  MoveL 4549 to (447.41, 537.05, 80) mm, rotated rx -180 ry 0 rz 160 deg; joints [12.233, 59.659, 9.495, -145.993, 72.482, 168.52]
  Set speed (17.8 mm/s)
  Call Extruder(266.02941)
  MoveL 4550 to (446.66, 535.95, 80) mm, rotated rx -180 ry 0 rz 160 deg; joints [12.104, 59.545, 9.763, -146.152, 72.584, 168.65]
  Call Extruder(270.12831)
  MoveL 4551 to (445.95, 534.87, 80) mm, rotated rx 180 ry 0 rz 160 deg; joints [11.975, 59.436, 10.019, -146.31, 72.681, 168.775]
  Set speed (17.8 mm/s)
  Call Extruder(274.24674)
  MoveL 4552 to (445.25, 533.77, 80) mm, rotated rx 180 ry 0 rz 160 deg; joints [11.843, 59.33, 10.27, -146.471, 72.776, 168.899]
  Call Extruder(278.37060)
  MoveL 4553 to (444.58, 532.66, 80) mm, rotated rx -180 ry 0 rz 160 deg; joints [11.707, 59.226, 10.515, -146.634, 72.867, 169.022]
  Set speed (17.8 mm/s)
  Call Extruder(282.63092)
  MoveL 4554 to (443.91, 531.49, 80) mm, rotated rx 180 ry 0 rz 160 deg; joints [11.563, 59.122, 10.76, -146.806, 72.959, 169.146]
  Call Extruder(286.74153)
  MoveL 4555 to (443.28, 530.35, 80) mm, rotated rx -180 ry 0 rz 160 deg; joints [11.421, 59.025, 10.991, -146.974, 73.044, 169.265]
  Call Extruder(290.93893)
  MoveL 4556 to (442.67, 529.17, 80) mm, rotated rx 180 ry 0 rz 160 deg; joints [11.274, 58.929, 11.219, -147.147, 73.127, 169.384]
  Set speed (17.8 mm/s)
  Call Extruder(295.04718)
  MoveL 4557 to (442.09, 528.01, 80) mm, rotated rx 180 ry 0 rz 160 deg; joints [11.126, 58.838, 11.436, -147.32, 73.205, 169.499]
  Set speed (17.8 mm/s)
  Call Extruder(299.35678)
  MoveL 4558 to (441.52, 526.78, 80) mm, rotated rx 180 ry 0 rz 160 deg; joints [10.968, 58.746, 11.654, -147.503, 73.283, 169.617]
  Set speed (17.8 mm/s)
  Call Extruder(303.33927)
  MoveL 4559 to (441, 525.63, 80) mm, rotated rx 180 ry 0 rz 160 deg; joints [10.82, 58.663, 11.851, -147.673, 73.353, 169.725]
  Set speed (17.8 mm/s)
  Call Extruder(307.68159)
  MoveL 4560 to (440.47, 524.37, 80) mm, rotated rx 180 ry 0 rz 160 deg; joints [10.654, 58.577, 12.056, -147.862, 73.424, 169.839]
  Set speed (17.8 mm/s)
  Call Extruder(311.65960)
  MoveL 4561 to (440, 523.2, 80) mm, rotated rx 180 ry 0 rz 160 deg; joints [10.501, 58.5, 12.239, -148.036, 73.488, 169.943]
  Set speed (17.8 mm/s)
  Call Extruder(316.02784)
  MoveL 4562 to (439.53, 521.91, 80) mm, rotated rx 180 ry 0 rz 160 deg; joints [10.33, 58.421, 12.429, -148.229, 73.552, 170.054]
  Call Extruder(320.19544)
  MoveL 4563 to (439.08, 520.67, 80) mm, rotated rx -180 ry 0 rz 160 deg; joints [10.164, 58.347, 12.607, -148.415, 73.612, 170.159]
  Set speed (17.8 mm/s)
  Call Extruder(324.35507)
  MoveL 4564 to (438.68, 519.42, 80) mm, rotated rx 180 ry 0 rz 160 deg; joints [9.996, 58.278, 12.773, -148.603, 73.665, 170.26]
  Call Extruder(328.30973)
  MoveL 4565 to (438.31, 518.23, 80) mm, rotated rx -180 ry 0 rz 160 deg; joints [9.834, 58.213, 12.926, -148.782, 73.715, 170.355]
  Call Extruder(332.69708)
  MoveL 4566 to (437.94, 516.9, 80) mm, rotated rx 180 ry 0 rz 160 deg; joints [9.652, 58.147, 13.086, -148.984, 73.764, 170.458]
  Set speed (17.8 mm/s)
  Call Extruder(336.73190)
  MoveL 4567 to (437.61, 515.67, 80) mm, rotated rx 180 ry 0 rz 160 deg; joints [9.483, 58.088, 13.227, -149.17, 73.807, 170.55]
  Set speed (17.8 mm/s)
  Call Extruder(341.04868)
  MoveL 4568 to (437.3, 514.34, 80) mm, rotated rx -180 ry 0 rz 160 deg; joints [9.299, 58.03, 13.368, -149.371, 73.848, 170.647]
  Call Extruder(345.11422)
  MoveL 4569 to (437.02, 513.09, 80) mm, rotated rx -180 ry 0 rz 160 deg; joints [9.125, 57.977, 13.496, -149.561, 73.884, 170.736]
  Set speed (17.8 mm/s)
  Call Extruder(353.56410)
  MoveL 4570 to (436.53, 510.46, 80) mm, rotated rx 180 ry 0 rz 160 deg; joints [8.756, 57.878, 13.734, -149.96, 73.946, 170.914]
  Set speed (17.8 mm/s)
  Call Extruder(361.89397)
  MoveL 4571 to (436.15, 507.86, 80) mm, rotated rx 180 ry 0 rz 160 deg; joints [8.386, 57.794, 13.937, -150.358, 73.991, 171.081]
  Call Extruder(370.22374)
  MoveL 4572 to (435.89, 505.24, 80) mm, rotated rx -180 ry 0 rz 160 deg; joints [8.01, 57.724, 14.107, -150.758, 74.02, 171.238]
  Set speed (17.8 mm/s)
  Call Extruder(378.39440)
  MoveL 4573 to (435.73, 502.67, 80) mm, rotated rx -180 ry 0 rz 160 deg; joints [7.637, 57.668, 14.242, -151.153, 74.033, 171.384]
  Set speed (17.8 mm/s)
  Call Extruder(386.80288)
  MoveL 4574 to (435.67, 500.01, 80) mm, rotated rx 180 ry 0 rz 160 deg; joints [7.249, 57.624, 14.348, -151.56, 74.03, 171.524]
  Set speed (17.8 mm/s)
  Call Extruder(394.37867)
  MoveL 4575 to (435.72, 497.62, 80) mm, rotated rx 180 ry 0 rz 160 deg; joints [6.897, 57.597, 14.415, -151.927, 74.013, 171.644]
  Set speed (17.8 mm/s)
  Call Extruder(401.68594)
  MoveL 4576 to (435.84, 495.31, 80) mm, rotated rx -180 ry 0 rz 160 deg; joints [6.557, 57.581, 14.453, -152.281, 73.984, 171.751]
  Set speed (17.8 mm/s)
  Call Extruder(409.27011)
  MoveL 4577 to (436.06, 492.92, 80) mm, rotated rx 180 ry 0 rz 160 deg; joints [6.203, 57.576, 14.465, -152.646, 73.94, 171.855]
  Set speed (17.8 mm/s)
  Call Extruder(416.76691)
  MoveL 4578 to (436.37, 490.57, 80) mm, rotated rx 180 ry 0 rz 160 deg; joints [5.853, 57.582, 14.451, -153.006, 73.883, 171.951]
  Set speed (17.8 mm/s)
  Call Extruder(424.33928)
  MoveL 4579 to (436.76, 488.21, 80) mm, rotated rx -180 ry 0 rz 160 deg; joints [5.5, 57.599, 14.408, -153.367, 73.811, 172.041]
  Set speed (17.8 mm/s)
  Call Extruder(431.68669)
  MoveL 4580 to (437.23, 485.94, 80) mm, rotated rx -180 ry 0 rz 160 deg; joints [5.159, 57.627, 14.341, -153.713, 73.729, 172.121]
  Call Extruder(439.23159)
  MoveL 4581 to (437.79, 483.62, 80) mm, rotated rx -180 ry 0 rz 160 deg; joints [4.811, 57.666, 14.245, -154.065, 73.631, 172.196]
  Set speed (17.8 mm/s)
  Call Extruder(446.63182)
  MoveL 4582 to (438.43, 481.37, 80) mm, rotated rx -180 ry 0 rz 160 deg; joints [4.472, 57.716, 14.125, -154.405, 73.522, 172.263]
  Call Extruder(454.15459)
  MoveL 4583 to (439.16, 479.11, 80) mm, rotated rx 180 ry 0 rz 160 deg; joints [4.132, 57.778, 13.976, -154.746, 73.397, 172.324]
  Set speed (17.8 mm/s)
  Call Extruder(461.75851)
  MoveL 4584 to (439.98, 476.85, 80) mm, rotated rx 180 ry 0 rz 160 deg; joints [3.793, 57.851, 13.799, -155.084, 73.258, 172.378]
  Call Extruder(469.29190)
  MoveL 4585 to (440.88, 474.64, 80) mm, rotated rx -180 ry 0 rz 160 deg; joints [3.461, 57.935, 13.597, -155.412, 73.107, 172.426]
  Set speed (17.8 mm/s)
  Call Extruder(476.78431)
  MoveL 4586 to (441.85, 472.48, 80) mm, rotated rx 180 ry 0 rz 160 deg; joints [3.138, 58.029, 13.37, -155.731, 72.943, 172.466]
  Set speed (17.8 mm/s)
  Call Extruder(484.18602)
  MoveL 4587 to (442.89, 470.39, 80) mm, rotated rx -180 ry 0 rz 160 deg; joints [2.824, 58.133, 13.12, -156.038, 72.769, 172.5]
  Set speed (17.8 mm/s)
  Call Extruder(491.62160)
  MoveL 4588 to (444.01, 468.32, 80) mm, rotated rx -180 ry 0 rz 160 deg; joints [2.516, 58.247, 12.845, -156.338, 72.582, 172.527]
  Set speed (17.8 mm/s)
  Call Extruder(499.11200)
  MoveL 4589 to (445.22, 466.28, 80) mm, rotated rx -180 ry 0 rz 160 deg; joints [2.212, 58.373, 12.543, -156.631, 72.381, 172.549]
  Set speed (17.8 mm/s)
  Call Extruder(506.66974)
  MoveL 4590 to (446.51, 464.27, 80) mm, rotated rx -180 ry 0 rz 160 deg; joints [1.915, 58.511, 12.214, -156.917, 72.166, 172.564]
  Set speed (17.8 mm/s)
  Call Extruder(514.00848)
  MoveL 4591 to (447.83, 462.37, 80) mm, rotated rx 180 ry 0 rz 160 deg; joints [1.633, 58.655, 11.871, -157.185, 71.947, 172.573]
  Call Extruder(521.73808)
  MoveL 4592 to (449.3, 460.41, 80) mm, rotated rx -180 ry 0 rz 160 deg; joints [1.347, 58.817, 11.485, -157.456, 71.703, 172.575]
  Set speed (17.8 mm/s)
  Call Extruder(529.07649)
  MoveL 4593 to (450.76, 458.61, 80) mm, rotated rx -180 ry 0 rz 160 deg; joints [1.084, 58.981, 11.096, -157.702, 71.461, 172.571]
  Set speed (17.8 mm/s)
  Call Extruder(536.63592)
  MoveL 4594 to (452.33, 456.81, 80) mm, rotated rx -180 ry 0 rz 160 deg; joints [0.823, 59.159, 10.673, -157.944, 71.201, 172.561]
  Set speed (17.8 mm/s)
  Call Extruder(544.21793)
  MoveL 4595 to (453.97, 455.06, 80) mm, rotated rx -180 ry 0 rz 160 deg; joints [0.571, 59.348, 10.227, -158.175, 70.93, 172.545]
  Call Extruder(551.61734)
  MoveL 4596 to (455.63, 453.42, 80) mm, rotated rx 180 ry 0 rz 160 deg; joints [0.337, 59.542, 9.769, -158.387, 70.655, 172.523]
  Set speed (17.8 mm/s)
  Call Extruder(559.11753)
  MoveL 4597 to (457.38, 451.82, 80) mm, rotated rx 180 ry 0 rz 160 deg; joints [0.109, 59.749, 9.285, -158.59, 70.366, 172.495]
  Call Extruder(566.69343)
  MoveL 4598 to (459.2, 450.27, 80) mm, rotated rx 180 ry 0 rz 160 deg; joints [-0.109, 59.967, 8.775, -158.782, 70.065, 172.46]
  Set speed (17.8 mm/s)
  Call Extruder(574.44703)
  MoveL 4599 to (461.12, 448.75, 80) mm, rotated rx -180 ry 0 rz 160 deg; joints [-0.32, 60.199, 8.233, -158.964, 69.749, 172.417]
  Set speed (17.8 mm/s)
  Call Extruder(581.05646)
  MoveL 4600 to (462.81, 447.51, 80) mm, rotated rx 180 ry 0 rz 160 deg; joints [-0.491, 60.404, 7.755, -159.108, 69.472, 172.376]
  Set speed (17.8 mm/s)
  Call Extruder(589.00388)
  MoveL 4601 to (464.88, 446.1, 80) mm, rotated rx -180 ry 0 rz 160 deg; joints [-0.683, 60.66, 7.16, -159.267, 69.13, 172.32]
  Set speed (17.8 mm/s)
  Call Extruder(596.68403)
  MoveL 4602 to (466.94, 444.82, 80) mm, rotated rx 180 ry 0 rz 160 deg; joints [-0.857, 60.917, 6.567, -159.406, 68.792, 172.259]
  Set speed (17.8 mm/s)
  Call Extruder(603.94088)
  MoveL 4603 to (468.93, 443.67, 80) mm, rotated rx 180 ry 0 rz 160 deg; joints [-1.009, 61.167, 5.99, -159.523, 68.465, 172.195]
  Call Extruder(611.62173)
  MoveL 4604 to (471.08, 442.54, 80) mm, rotated rx -180 ry 0 rz 160 deg; joints [-1.159, 61.44, 5.363, -159.633, 68.113, 172.121]
  Set speed (17.8 mm/s)
  Call Extruder(619.12505)
  MoveL 4605 to (473.21, 441.52, 80) mm, rotated rx -180 ry 0 rz 160 deg; joints [-1.292, 61.715, 4.734, -159.725, 67.762, 172.041]
  Call Extruder(626.65740)
  MoveL 4606 to (475.39, 440.56, 80) mm, rotated rx 180 ry 0 rz 160 deg; joints [-1.414, 61.998, 4.088, -159.804, 67.405, 171.955]
  Set speed (17.8 mm/s)
  Call Extruder(634.02253)
  MoveL 4607 to (477.56, 439.71, 80) mm, rotated rx -180 ry 0 rz 160 deg; joints [-1.52, 62.282, 3.442, -159.866, 67.049, 171.864]
  Set speed (17.8 mm/s)
  Call Extruder(641.66962)
  MoveL 4608 to (479.84, 438.91, 80) mm, rotated rx 180 ry 0 rz 160 deg; joints [-1.619, 62.584, 2.757, -159.916, 66.676, 171.763]
  Set speed (17.8 mm/s)
  Call Extruder(649.01644)
  MoveL 4609 to (482.05, 438.23, 80) mm, rotated rx 180 ry 0 rz 160 deg; joints [-1.702, 62.88, 2.087, -159.95, 66.313, 171.659]
  Set speed (17.8 mm/s)
  Call Extruder(656.55327)
  MoveL 4610 to (484.35, 437.61, 80) mm, rotated rx 180 ry 0 rz 160 deg; joints [-1.775, 63.191, 1.388, -159.97, 65.937, 171.545]
  Set speed (17.8 mm/s)
  Call Extruder(664.14451)
  MoveL 4611 to (486.69, 437.06, 80) mm, rotated rx -180 ry 0 rz 160 deg; joints [-1.836, 63.51, 0.671, -159.975, 65.555, 171.423]
  Call Extruder(671.49805)
  MoveL 4612 to (488.97, 436.63, 80) mm, rotated rx 180 ry 0 rz 160 deg; joints [-1.884, 63.824, -0.033, -159.966, 65.181, 171.298]
  Set speed (17.8 mm/s)
  Call Extruder(678.81827)
  MoveL 4613 to (491.26, 436.27, 80) mm, rotated rx 180 ry 0 rz 160 deg; joints [-1.921, 64.143, -0.744, -159.943, 64.807, 171.167]
  Call Extruder(686.41962)
  MoveL 4614 to (493.64, 435.99, 80) mm, rotated rx -180 ry 0 rz 160 deg; joints [-1.947, 64.479, -1.491, -159.904, 64.417, 171.022]
  Set speed (17.8 mm/s)
  Call Extruder(694.03784)
  MoveL 4615 to (496.04, 435.8, 80) mm, rotated rx -180 ry 0 rz 160 deg; joints [-1.961, 64.82, -2.248, -159.851, 64.024, 170.87]
  Set speed (17.8 mm/s)
  Call Extruder(701.60500)
  MoveL 4616 to (498.43, 435.69, 80) mm, rotated rx 180 ry 0 rz 160 deg; joints [-1.964, 65.164, -3.007, -159.784, 63.633, 170.712]
  Set speed (17.8 mm/s)
  Call Extruder(709.02942)
  MoveL 4617 to (500.78, 435.68, 80) mm, rotated rx 180 ry 0 rz 160 deg; joints [-1.955, 65.505, -3.759, -159.703, 63.249, 170.549]
  Set speed (17.9 mm/s)
  Call Extruder(716.40203)
  MoveL 4618 to (503.11, 435.75, 80) mm, rotated rx -180 ry 0 rz 160 deg; joints [-1.936, 65.847, -4.512, -159.61, 62.868, 170.379]
  Set speed (17.9 mm/s)
  Call Extruder(724.01110)
  MoveL 4619 to (505.51, 435.91, 80) mm, rotated rx -180 ry 0 rz 160 deg; joints [-1.906, 66.204, -5.295, -159.499, 62.475, 170.196]
  Set speed (17.8 mm/s)
  Call Extruder(731.57340)
  MoveL 4620 to (507.89, 436.16, 80) mm, rotated rx -180 ry 0 rz 160 deg; joints [-1.865, 66.562, -6.076, -159.375, 62.085, 170.007]
  Set speed (17.8 mm/s)
  Call Extruder(738.91714)
  MoveL 4621 to (510.19, 436.49, 80) mm, rotated rx 180 ry 0 rz 160 deg; joints [-1.815, 66.911, -6.837, -159.242, 61.709, 169.816]
  Set speed (17.8 mm/s)
  Call Extruder(746.32248)
  MoveL 4622 to (512.49, 436.9, 80) mm, rotated rx 180 ry 0 rz 160 deg; joints [-1.755, 67.266, -7.607, -159.094, 61.331, 169.616]
  Set speed (17.8 mm/s)
  Call Extruder(753.98830)
  MoveL 4623 to (514.86, 437.41, 80) mm, rotated rx -180 ry 0 rz 160 deg; joints [-1.682, 67.635, -8.406, -158.928, 60.943, 169.4]
  Set speed (17.8 mm/s)
  Call Extruder(761.38063)
  MoveL 4624 to (517.12, 437.99, 80) mm, rotated rx 180 ry 0 rz 160 deg; joints [-1.603, 67.992, -9.177, -158.755, 60.571, 169.185]
  Call Extruder(769.10386)
  MoveL 4625 to (519.47, 438.69, 80) mm, rotated rx -180 ry 0 rz 160 deg; joints [-1.51, 68.365, -9.982, -158.561, 60.187, 168.953]
  Set speed (17.8 mm/s)
  Call Extruder(776.51579)
  MoveL 4626 to (521.68, 439.44, 80) mm, rotated rx 180 ry 0 rz 160 deg; joints [-1.412, 68.724, -10.753, -158.362, 59.822, 168.722]
  Call Extruder(783.77355)
  MoveL 4627 to (523.83, 440.25, 80) mm, rotated rx 180 ry 0 rz 160 deg; joints [-1.307, 69.076, -11.506, -158.156, 59.47, 168.49]
  Set speed (17.8 mm/s)
  Call Extruder(791.50170)
  MoveL 4628 to (526.08, 441.2, 80) mm, rotated rx 180 ry 0 rz 160 deg; joints [-1.187, 69.449, -12.305, -157.924, 59.1, 168.235]
  Call Extruder(798.99684)
  MoveL 4629 to (528.23, 442.2, 80) mm, rotated rx -180 ry 0 rz 160 deg; joints [-1.061, 69.81, -13.075, -157.688, 58.747, 167.981]
  Call Extruder(806.41157)
  MoveL 4630 to (530.31, 443.26, 80) mm, rotated rx 180 ry 0 rz 160 deg; joints [-0.929, 70.166, -13.832, -157.443, 58.404, 167.722]
  Set speed (17.8 mm/s)
  Call Extruder(813.98236)
  MoveL 4631 to (532.4, 444.43, 80) mm, rotated rx 180 ry 0 rz 160 deg; joints [-0.787, 70.527, -14.599, -157.183, 58.06, 167.452]
  Set speed (17.8 mm/s)
  Call Extruder(821.38405)
  MoveL 4632 to (534.4, 445.64, 80) mm, rotated rx -180 ry 0 rz 160 deg; joints [-0.639, 70.878, -15.341, -156.917, 57.732, 167.181]
  Set speed (17.8 mm/s)
  Call Extruder(828.97367)
  MoveL 4633 to (536.41, 446.97, 80) mm, rotated rx 180 ry 0 rz 160 deg; joints [-0.481, 71.234, -16.095, -156.635, 57.402, 166.898]
  Set speed (17.8 mm/s)
  Call Extruder(836.31752)
  MoveL 4634 to (538.3, 448.31, 80) mm, rotated rx -180 ry 0 rz 160 deg; joints [-0.321, 71.575, -16.814, -156.352, 57.092, 166.618]
  Set speed (17.8 mm/s)
  Call Extruder(843.95014)
  MoveL 4635 to (540.21, 449.79, 80) mm, rotated rx 180 ry 0 rz 160 deg; joints [-0.147, 71.926, -17.552, -156.049, 56.778, 166.322]
  Set speed (17.8 mm/s)
  Call Extruder(851.24676)
  MoveL 4636 to (541.98, 451.26, 80) mm, rotated rx -180 ry 0 rz 160 deg; joints [0.025, 72.256, -18.246, -155.751, 56.488, 166.034]
  Set speed (17.8 mm/s)
  Call Extruder(858.93004)
  MoveL 4637 to (543.79, 452.88, 80) mm, rotated rx -180 ry 0 rz 160 deg; joints [0.213, 72.599, -18.964, -155.428, 56.192, 165.726]
  Call Extruder(866.36806)
  MoveL 4638 to (545.49, 454.51, 80) mm, rotated rx 180 ry 0 rz 160 deg; joints [0.402, 72.924, -19.646, -155.108, 55.915, 165.424]
  Set speed (17.8 mm/s)
  Call Extruder(870.44520)
  MoveL 4639 to (546.39, 455.43, 80) mm, rotated rx -180 ry 0 rz 160 deg; joints [0.507, 73.1, -20.012, -154.93, 55.769, 165.257]
  Set speed (17.8 mm/s)
  Call Extruder(874.59411)
  MoveL 4640 to (547.29, 456.39, 80) mm, rotated rx 180 ry 0 rz 160 deg; joints [0.617, 73.277, -20.381, -154.746, 55.623, 165.086]
  Set speed (17.8 mm/s)
  Call Extruder(878.97391)
  MoveL 4641 to (548.22, 457.42, 80) mm, rotated rx 180 ry 0 rz 160 deg; joints [0.734, 73.461, -20.766, -154.55, 55.472, 164.904]
  Set speed (17.8 mm/s)
  Call Extruder(883.03818)
  MoveL 4642 to (549.06, 458.39, 80) mm, rotated rx -180 ry 0 rz 160 deg; joints [0.844, 73.63, -21.117, -154.366, 55.336, 164.735]
  Set speed (17.8 mm/s)
  Call Extruder(887.06977)
  MoveL 4643 to (549.87, 459.37, 80) mm, rotated rx 180 ry 0 rz 160 deg; joints [0.956, 73.794, -21.46, -154.182, 55.205, 164.566]
  Set speed (17.9 mm/s)
  Call Extruder(891.22700)
  MoveL 4644 to (550.69, 460.4, 80) mm, rotated rx -180 ry 0 rz 160 deg; joints [1.072, 73.962, -21.809, -153.991, 55.074, 164.392]
  Call Extruder(895.38513)
  MoveL 4645 to (551.49, 461.44, 80) mm, rotated rx 180 ry 0 rz 160 deg; joints [1.189, 74.127, -22.152, -153.797, 54.946, 164.217]
  Set speed (17.8 mm/s)
  Call Extruder(899.59619)
  MoveL 4646 to (552.28, 462.51, 80) mm, rotated rx 180 ry 0 rz 160 deg; joints [1.31, 74.291, -22.493, -153.6, 54.82, 164.04]
  Set speed (17.8 mm/s)
  Call Extruder(903.72520)
  MoveL 4647 to (553.03, 463.58, 80) mm, rotated rx -180 ry 0 rz 160 deg; joints [1.43, 74.449, -22.821, -153.406, 54.701, 163.866]
  Set speed (17.8 mm/s)
  Call Extruder(907.95576)
  MoveL 4648 to (553.77, 464.69, 80) mm, rotated rx 180 ry 0 rz 160 deg; joints [1.554, 74.609, -23.151, -153.205, 54.584, 163.687]
  Set speed (17.8 mm/s)
  Call Extruder(912.06776)
  MoveL 4649 to (554.48, 465.79, 80) mm, rotated rx -180 ry 0 rz 160 deg; joints [1.676, 74.76, -23.464, -153.009, 54.474, 163.513]
  Call Extruder(916.21351)
  MoveL 4650 to (555.16, 466.9, 80) mm, rotated rx -180 ry 0 rz 160 deg; joints [1.801, 74.91, -23.774, -152.81, 54.367, 163.338]
  Set speed (17.8 mm/s)
  Call Extruder(920.42391)
  MoveL 4651 to (555.83, 468.05, 80) mm, rotated rx 180 ry 0 rz 160 deg; joints [1.929, 75.058, -24.08, -152.607, 54.263, 163.161]
  Set speed (17.8 mm/s)
  Call Extruder(925.81268)
  MoveL 4652 to (556.66, 469.54, 80) mm, rotated rx -180 ry 0 rz 160 deg; joints [2.094, 75.243, -24.463, -152.347, 54.136, 162.935]
  Set speed (17.8 mm/s)
  Call Extruder(928.72194)
  MoveL 4653 to (557.09, 470.35, 80) mm, rotated rx -180 ry 0 rz 160 deg; joints [2.184, 75.34, -24.663, -152.206, 54.071, 162.813]
  Set speed (17.8 mm/s)
  Call Extruder(932.89329)
  MoveL 4654 to (557.68, 471.53, 80) mm, rotated rx 180 ry 0 rz 160 deg; joints [2.314, 75.477, -24.946, -152.003, 53.981, 162.639]
  Call Extruder(938.19287)
  MoveL 4655 to (558.41, 473.04, 80) mm, rotated rx 180 ry 0 rz 160 deg; joints [2.481, 75.646, -25.295, -151.745, 53.872, 162.418]
  Call Extruder(941.26626)
  MoveL 4656 to (558.81, 473.92, 80) mm, rotated rx -180 ry 0 rz 160 deg; joints [2.579, 75.74, -25.488, -151.595, 53.815, 162.292]
  Set speed (17.8 mm/s)
  Call Extruder(945.43897)
  MoveL 4657 to (559.32, 475.14, 80) mm, rotated rx 180 ry 0 rz 160 deg; joints [2.712, 75.864, -25.743, -151.391, 53.74, 162.121]
  Set speed (17.8 mm/s)
  Call Extruder(949.41645)
  MoveL 4658 to (559.8, 476.3, 80) mm, rotated rx 180 ry 0 rz 160 deg; joints [2.84, 75.981, -25.983, -151.197, 53.671, 161.958]
  Set speed (17.8 mm/s)
  Call Extruder(953.76538)
  MoveL 4659 to (560.29, 477.58, 80) mm, rotated rx 180 ry 0 rz 160 deg; joints [2.981, 76.101, -26.231, -150.985, 53.604, 161.783]
  Call Extruder(957.86713)
  MoveL 4660 to (560.73, 478.8, 80) mm, rotated rx -180 ry 0 rz 160 deg; joints [3.115, 76.213, -26.461, -150.785, 53.543, 161.618]
  Set speed (17.8 mm/s)
  Call Extruder(962.11224)
  MoveL 4661 to (561.15, 480.07, 80) mm, rotated rx -180 ry 0 rz 160 deg; joints [3.255, 76.322, -26.684, -150.578, 53.487, 161.45]
  Call Extruder(966.43379)
  MoveL 4662 to (561.57, 481.37, 80) mm, rotated rx 180 ry 0 rz 160 deg; joints [3.397, 76.431, -26.908, -150.368, 53.433, 161.279]
  Set speed (17.8 mm/s)
  Call Extruder(970.44890)
  MoveL 4663 to (561.92, 482.59, 80) mm, rotated rx 180 ry 0 rz 160 deg; joints [3.531, 76.525, -27.101, -150.174, 53.39, 161.124]
  Call Extruder(974.61044)
  MoveL 4664 to (562.27, 483.85, 80) mm, rotated rx -180 ry 0 rz 160 deg; joints [3.67, 76.621, -27.297, -149.973, 53.348, 160.964]
  Set speed (17.8 mm/s)
  Call Extruder(982.89558)
  MoveL 4665 to (562.88, 486.4, 80) mm, rotated rx -180 ry 0 rz 160 deg; joints [3.949, 76.795, -27.655, -149.575, 53.281, 160.653]
  Call Extruder(991.08728)
  MoveL 4666 to (563.37, 488.94, 80) mm, rotated rx 180 ry 0 rz 160 deg; joints [4.228, 76.948, -27.968, -149.186, 53.236, 160.354]
  Set speed (17.8 mm/s)
  Call Extruder(999.56666)
  MoveL 4667 to (563.78, 491.59, 80) mm, rotated rx 180 ry 0 rz 160 deg; joints [4.519, 77.087, -28.252, -148.789, 53.21, 160.056]
  Set speed (17.9 mm/s)
  Call Extruder(1007.97979)
  MoveL 4668 to (564.07, 494.23, 80) mm, rotated rx 180 ry 0 rz 160 deg; joints [4.809, 77.203, -28.491, -148.4, 53.206, 159.773]
  Call Extruder(1016.20362)
  MoveL 4669 to (564.25, 496.83, 80) mm, rotated rx 180 ry 0 rz 160 deg; joints [5.095, 77.297, -28.682, -148.028, 53.222, 159.508]
  Call Extruder(1024.53113)
  MoveL 4670 to (564.33, 499.46, 80) mm, rotated rx 180 ry 0 rz 160 deg; joints [5.386, 77.37, -28.831, -147.658, 53.26, 159.255]
  Set speed (17.8 mm/s)
  Call Extruder(1032.73408)
  MoveL 4671 to (564.29, 502.06, 80) mm, rotated rx 180 ry 0 rz 160 deg; joints [5.673, 77.421, -28.935, -147.302, 53.317, 159.019]
  Set speed (17.8 mm/s)
  Call Extruder(1041.16777)
  MoveL 4672 to (564.16, 504.72, 80) mm, rotated rx 180 ry 0 rz 160 deg; joints [5.968, 77.451, -28.998, -146.945, 53.397, 158.792]
  Call Extruder(1049.40798)
  MoveL 4673 to (563.91, 507.31, 80) mm, rotated rx 180 ry 0 rz 160 deg; joints [6.257, 77.459, -29.014, -146.607, 53.495, 158.587]
  Call Extruder(1057.90097)
  MoveL 4674 to (563.55, 509.97, 80) mm, rotated rx 180 ry 0 rz 160 deg; joints [6.555, 77.445, -28.985, -146.268, 53.617, 158.392]
  Set speed (17.8 mm/s)
  Call Extruder(1066.13070)
  MoveL 4675 to (563.1, 512.53, 80) mm, rotated rx -180 ry 0 rz 160 deg; joints [6.844, 77.409, -28.912, -145.951, 53.754, 158.221]
  Set speed (17.8 mm/s)
  Call Extruder(1074.27794)
  MoveL 4676 to (562.54, 515.05, 80) mm, rotated rx -180 ry 0 rz 160 deg; joints [7.128, 77.353, -28.797, -145.648, 53.909, 158.069]
  Set speed (17.8 mm/s)
  Call Extruder(1078.65148)
  MoveL 4677 to (562.2, 516.39, 80) mm, rotated rx 180 ry 0 rz 160 deg; joints [7.281, 77.312, -28.714, -145.49, 54.001, 157.996]
  Set speed (17.8 mm/s)
  Call Extruder(1082.98970)
  MoveL 4678 to (561.84, 517.71, 80) mm, rotated rx -180 ry 0 rz 160 deg; joints [7.432, 77.27, -28.627, -145.336, 54.094, 157.925]
  Set speed (17.8 mm/s)
  Call Extruder(1091.00038)
  MoveL 4679 to (561.1, 520.13, 80) mm, rotated rx -180 ry 0 rz 160 deg; joints [7.709, 77.173, -28.429, -145.06, 54.282, 157.811]
  Set speed (17.8 mm/s)
  Call Extruder(1095.29692)
  MoveL 4680 to (560.65, 521.41, 80) mm, rotated rx 180 ry 0 rz 160 deg; joints [7.857, 77.111, -28.303, -144.918, 54.39, 157.758]
  Set speed (17.8 mm/s)
  Call Extruder(1099.59245)
  MoveL 4681 to (560.19, 522.69, 80) mm, rotated rx 180 ry 0 rz 160 deg; joints [8.005, 77.048, -28.174, -144.777, 54.501, 157.707]
  Call Extruder(1103.62635)
  MoveL 4682 to (559.73, 523.88, 80) mm, rotated rx 180 ry 0 rz 160 deg; joints [8.143, 76.981, -28.035, -144.65, 54.611, 157.667]
  Call Extruder(1107.90082)
  MoveL 4683 to (559.22, 525.13, 80) mm, rotated rx 180 ry 0 rz 160 deg; joints [8.289, 76.907, -27.884, -144.516, 54.729, 157.626]
  Set speed (17.8 mm/s)
  Call Extruder(1111.96817)
  MoveL 4684 to (558.7, 526.3, 80) mm, rotated rx -180 ry 0 rz 160 deg; joints [8.427, 76.829, -27.724, -144.393, 54.848, 157.594]
  Set speed (17.8 mm/s)
  Call Extruder(1116.02326)
  MoveL 4685 to (558.17, 527.47, 80) mm, rotated rx 180 ry 0 rz 160 deg; joints [8.564, 76.749, -27.562, -144.272, 54.968, 157.564]
  Set speed (17.8 mm/s)
  Call Extruder(1120.19096)
  MoveL 4686 to (557.6, 528.65, 80) mm, rotated rx -180 ry 0 rz 160 deg; joints [8.705, 76.661, -27.381, -144.151, 55.097, 157.539]
  Set speed (17.9 mm/s)
  Call Extruder(1124.37462)
  MoveL 4687 to (556.99, 529.83, 80) mm, rotated rx 180 ry 0 rz 160 deg; joints [8.846, 76.569, -27.191, -144.033, 55.23, 157.519]
  Set speed (17.8 mm/s)
  Call Extruder(1128.55393)
  MoveL 4688 to (556.37, 531, 80) mm, rotated rx -180 ry 0 rz 160 deg; joints [8.985, 76.471, -26.99, -143.918, 55.366, 157.503]
  Set speed (17.8 mm/s)
  Call Extruder(1132.80711)
  MoveL 4689 to (555.71, 532.16, 80) mm, rotated rx 180 ry 0 rz 160 deg; joints [9.126, 76.367, -26.776, -143.805, 55.509, 157.492]
  Set speed (17.8 mm/s)
  Call Extruder(1137.78181)
  MoveL 4690 to (554.91, 533.52, 80) mm, rotated rx -180 ry 0 rz 160 deg; joints [9.29, 76.24, -26.516, -143.675, 55.679, 157.484]
  Set speed (17.8 mm/s)
  Call Extruder(1141.04464)
  MoveL 4691 to (554.36, 534.39, 80) mm, rotated rx -180 ry 0 rz 160 deg; joints [9.397, 76.153, -26.337, -143.593, 55.794, 157.483]
  Call Extruder(1144.61353)
  MoveL 4692 to (553.75, 535.34, 80) mm, rotated rx 180 ry 0 rz 160 deg; joints [9.513, 76.054, -26.134, -143.505, 55.923, 157.484]
  Call Extruder(1149.35669)
  MoveL 4693 to (552.92, 536.58, 80) mm, rotated rx 180 ry 0 rz 160 deg; joints [9.666, 75.919, -25.857, -143.392, 56.096, 157.491]
  Set speed (17.8 mm/s)
  Call Extruder(1153.55545)
  MoveL 4694 to (552.15, 537.67, 80) mm, rotated rx 180 ry 0 rz 160 deg; joints [9.801, 75.795, -25.601, -143.294, 56.253, 157.502]
  Call Extruder(1157.83743)
  MoveL 4695 to (551.35, 538.75, 80) mm, rotated rx 180 ry 0 rz 160 deg; joints [9.938, 75.664, -25.332, -143.198, 56.416, 157.518]
  Set speed (17.8 mm/s)
  Call Extruder(1161.84532)
  MoveL 4696 to (550.57, 539.76, 80) mm, rotated rx 180 ry 0 rz 160 deg; joints [10.064, 75.538, -25.072, -143.111, 56.571, 157.537]
  Set speed (17.8 mm/s)
  Call Extruder(1166.05691)
  MoveL 4697 to (549.74, 540.8, 80) mm, rotated rx 180 ry 0 rz 160 deg; joints [10.196, 75.402, -24.79, -143.022, 56.738, 157.561]
  Set speed (17.8 mm/s)
  Call Extruder(1170.18772)
  MoveL 4698 to (548.9, 541.8, 80) mm, rotated rx 180 ry 0 rz 160 deg; joints [10.324, 75.264, -24.507, -142.938, 56.904, 157.589]
  Set speed (17.8 mm/s)
  Call Extruder(1174.31180)
  MoveL 4699 to (548.04, 542.78, 80) mm, rotated rx 180 ry 0 rz 160 deg; joints [10.451, 75.124, -24.217, -142.857, 57.071, 157.62]
  Call Extruder(1178.49581)
  MoveL 4700 to (547.15, 543.76, 80) mm, rotated rx -180 ry 0 rz 160 deg; joints [10.579, 74.978, -23.915, -142.777, 57.244, 157.656]
  Set speed (17.8 mm/s)
  Call Extruder(1182.67813)
  MoveL 4701 to (546.25, 544.72, 80) mm, rotated rx 180 ry 0 rz 160 deg; joints [10.705, 74.829, -23.606, -142.701, 57.419, 157.696]
  Call Extruder(1186.85012)
  MoveL 4702 to (545.32, 545.66, 80) mm, rotated rx 180 ry 0 rz 160 deg; joints [10.829, 74.677, -23.291, -142.627, 57.595, 157.739]
  Set speed (17.8 mm/s)
  Call Extruder(1190.99617)
  MoveL 4703 to (544.38, 546.57, 80) mm, rotated rx 180 ry 0 rz 160 deg; joints [10.952, 74.522, -22.971, -142.557, 57.773, 157.787]
  Set speed (17.8 mm/s)
  Call Extruder(1195.13887)
  MoveL 4704 to (543.42, 547.46, 80) mm, rotated rx 180 ry 0 rz 160 deg; joints [11.073, 74.365, -22.645, -142.489, 57.953, 157.838]
  Set speed (17.8 mm/s)
  Call Extruder(1199.32285)
  MoveL 4705 to (542.44, 548.35, 80) mm, rotated rx 180 ry 0 rz 160 deg; joints [11.193, 74.203, -22.308, -142.423, 58.136, 157.893]
  Call Extruder(1203.51241)
  MoveL 4706 to (541.43, 549.21, 80) mm, rotated rx -180 ry 0 rz 160 deg; joints [11.312, 74.038, -21.966, -142.361, 58.322, 157.953]
  Set speed (17.8 mm/s)
  Call Extruder(1207.76800)
  MoveL 4707 to (540.39, 550.07, 80) mm, rotated rx -180 ry 0 rz 160 deg; joints [11.432, 73.867, -21.612, -142.299, 58.512, 158.016]
  Call Extruder(1211.79044)
  MoveL 4708 to (539.4, 550.85, 80) mm, rotated rx -180 ry 0 rz 160 deg; joints [11.544, 73.704, -21.272, -142.244, 58.694, 158.08]
  Set speed (17.8 mm/s)
  Call Extruder(1215.97259)
  MoveL 4709 to (538.34, 551.65, 80) mm, rotated rx -180 ry 0 rz 160 deg; joints [11.658, 73.532, -20.913, -142.189, 58.884, 158.149]
  Set speed (17.8 mm/s)
  Call Extruder(1220.15658)
  MoveL 4710 to (537.27, 552.43, 80) mm, rotated rx -180 ry 0 rz 160 deg; joints [11.771, 73.357, -20.549, -142.137, 59.075, 158.222]
  Set speed (17.8 mm/s)
  Call Extruder(1224.28353)
  MoveL 4711 to (536.2, 553.18, 80) mm, rotated rx 180 ry 0 rz 160 deg; joints [11.88, 73.182, -20.184, -142.088, 59.266, 158.297]
  Call Extruder(1228.44477)
  MoveL 4712 to (535.11, 553.9, 80) mm, rotated rx 180 ry 0 rz 160 deg; joints [11.989, 73.004, -19.811, -142.042, 59.459, 158.376]
  Set speed (17.8 mm/s)
  Call Extruder(1232.73871)
  MoveL 4713 to (533.96, 554.63, 80) mm, rotated rx -180 ry 0 rz 160 deg; joints [12.099, 72.817, -19.421, -141.997, 59.66, 158.461]
  Set speed (17.8 mm/s)
  Call Extruder(1237.59762)
  MoveL 4714 to (532.65, 555.43, 80) mm, rotated rx -180 ry 0 rz 160 deg; joints [12.221, 72.604, -18.976, -141.948, 59.888, 158.56]
  Set speed (17.8 mm/s)
  Call Extruder(1241.01631)
  MoveL 4715 to (531.72, 555.97, 80) mm, rotated rx 180 ry 0 rz 160 deg; joints [12.306, 72.453, -18.659, -141.916, 60.049, 158.633]
  Set speed (17.8 mm/s)
  Call Extruder(1244.53094)
  MoveL 4716 to (530.75, 556.51, 80) mm, rotated rx -180 ry 0 rz 160 deg; joints [12.391, 72.296, -18.33, -141.885, 60.216, 158.709]
  Set speed (17.8 mm/s)
  Call Extruder(1250.50209)
  MoveL 4717 to (529.08, 557.39, 80) mm, rotated rx 180 ry 0 rz 160 deg; joints [12.534, 72.027, -17.765, -141.837, 60.5, 158.844]
  Set speed (17.8 mm/s)
  Call Extruder(1253.56154)
  MoveL 4718 to (528.21, 557.81, 80) mm, rotated rx 180 ry 0 rz 160 deg; joints [12.605, 71.887, -17.471, -141.815, 60.647, 158.916]
  Set speed (17.8 mm/s)
  Call Extruder(1257.72659)
  MoveL 4719 to (527.02, 558.38, 80) mm, rotated rx 180 ry 0 rz 160 deg; joints [12.7, 71.696, -17.069, -141.786, 60.847, 159.016]
  Set speed (17.8 mm/s)
  Call Extruder(1261.84604)
  MoveL 4720 to (525.83, 558.91, 80) mm, rotated rx -180 ry 0 rz 160 deg; joints [12.791, 71.506, -16.668, -141.761, 61.045, 159.118]
  Set speed (17.8 mm/s)
  Call Extruder(1266.00505)
  MoveL 4721 to (524.63, 559.43, 80) mm, rotated rx 180 ry 0 rz 160 deg; joints [12.883, 71.313, -16.262, -141.736, 61.245, 159.221]
  Call Extruder(1270.17478)
  MoveL 4722 to (523.4, 559.91, 80) mm, rotated rx -180 ry 0 rz 160 deg; joints [12.971, 71.118, -15.85, -141.716, 61.446, 159.33]
  Call Extruder(1274.35725)
  MoveL 4723 to (522.17, 560.39, 80) mm, rotated rx 180 ry 0 rz 160 deg; joints [13.058, 70.922, -15.436, -141.696, 61.648, 159.439]
  Set speed (17.8 mm/s)
  Call Extruder(1282.55297)
  MoveL 4724 to (519.72, 561.23, 80) mm, rotated rx -180 ry 0 rz 160 deg; joints [13.222, 70.534, -14.614, -141.666, 62.046, 159.662]
  Set speed (17.8 mm/s)
  Call Extruder(1287.61117)
  MoveL 4725 to (518.19, 561.7, 80) mm, rotated rx -180 ry 0 rz 160 deg; joints [13.317, 70.293, -14.103, -141.653, 62.291, 159.804]
  Set speed (17.8 mm/s)
  Call Extruder(1290.86870)
  MoveL 4726 to (517.21, 561.99, 80) mm, rotated rx -180 ry 0 rz 160 deg; joints [13.378, 70.138, -13.773, -141.645, 62.449, 159.897]
  Set speed (17.8 mm/s)
  Call Extruder(1294.63906)
  MoveL 4727 to (516.05, 562.29, 80) mm, rotated rx 180 ry 0 rz 160 deg; joints [13.445, 69.957, -13.388, -141.64, 62.632, 160.007]
  Set speed (17.8 mm/s)
  Call Extruder(1299.19985)
  MoveL 4728 to (514.66, 562.64, 80) mm, rotated rx 180 ry 0 rz 160 deg; joints [13.525, 69.739, -12.923, -141.635, 62.853, 160.141]
  Set speed (17.8 mm/s)
  Call Extruder(1307.67590)
  MoveL 4729 to (512.04, 563.19, 80) mm, rotated rx -180 ry 0 rz 160 deg; joints [13.664, 69.33, -12.051, -141.634, 63.263, 160.397]
  Set speed (17.8 mm/s)
  Call Extruder(1316.05487)
  MoveL 4730 to (509.43, 563.63, 80) mm, rotated rx 180 ry 0 rz 160 deg; joints [13.791, 68.925, -11.184, -141.643, 63.667, 160.657]
  Set speed (17.8 mm/s)
  Call Extruder(1324.22127)
  MoveL 4731 to (506.87, 563.96, 80) mm, rotated rx 180 ry 0 rz 160 deg; joints [13.904, 68.53, -10.336, -141.663, 64.06, 160.918]
  Set speed (17.8 mm/s)
  Call Extruder(1332.68330)
  MoveL 4732 to (504.21, 564.19, 80) mm, rotated rx 180 ry 0 rz 160 deg; joints [14.01, 68.12, -9.454, -141.692, 64.464, 161.195]
  Set speed (17.8 mm/s)
  Call Extruder(1341.05569)
  MoveL 4733 to (501.56, 564.31, 80) mm, rotated rx -180 ry 0 rz 160 deg; joints [14.103, 67.716, -8.581, -141.732, 64.862, 161.474]
  Call Extruder(1349.21391)
  MoveL 4734 to (498.98, 564.32, 80) mm, rotated rx -180 ry 0 rz 160 deg; joints [14.182, 67.323, -7.731, -141.781, 65.246, 161.752]
  Set speed (10.0 mm/s)
  MoveL 4735 to (498.98, 564.32, 84) mm, rotated rx 180 ry 0 rz 160 deg; joints [14.182, 66.666, -7.383, -141.693, 65.004, 161.541]
  Set speed (120.0 mm/s)
  MoveL 4736 to (498.95, 564.81, 84) mm, rotated rx -180 ry 0 rz 160 deg; joints [14.241, 66.68, -7.413, -141.626, 65.01, 161.503]
  Set speed (17.9 mm/s)
  Call Extruder(1357.64089)
  MoveL 4737 to (496.28, 564.71, 84) mm, rotated rx 180 ry 0 rz 160 deg; joints [14.311, 66.274, -6.536, -141.687, 65.401, 161.794]
  Set speed (17.9 mm/s)
  Call Extruder(1366.04197)
  MoveL 4738 to (493.63, 564.5, 84) mm, rotated rx 180 ry 0 rz 160 deg; joints [14.368, 65.872, -5.665, -141.76, 65.787, 162.089]
  Set speed (17.9 mm/s)
  Call Extruder(1374.34569)
  MoveL 4739 to (491.02, 564.19, 84) mm, rotated rx 180 ry 0 rz 160 deg; joints [14.412, 65.477, -4.807, -141.841, 66.164, 162.383]
  Set speed (17.9 mm/s)
  Call Extruder(1382.61213)
  MoveL 4740 to (488.43, 563.77, 84) mm, rotated rx -180 ry 0 rz 160 deg; joints [14.443, 65.088, -3.958, -141.934, 66.535, 162.68]
  Set speed (17.9 mm/s)
  Call Extruder(1391.15082)
  MoveL 4741 to (485.78, 563.24, 84) mm, rotated rx -180 ry 0 rz 160 deg; joints [14.461, 64.69, -3.088, -142.04, 66.912, 162.989]
  Set speed (17.9 mm/s)
  Call Extruder(1395.28127)
  MoveL 4742 to (484.5, 562.93, 84) mm, rotated rx 180 ry 0 rz 160 deg; joints [14.463, 64.499, -2.671, -142.097, 67.092, 163.14]
  Call Extruder(1399.32042)
  MoveL 4743 to (483.26, 562.62, 84) mm, rotated rx -180 ry 0 rz 160 deg; joints [14.464, 64.314, -2.265, -142.153, 67.267, 163.287]
  Set speed (17.9 mm/s)
  Call Extruder(1403.61831)
  MoveL 4744 to (481.96, 562.25, 84) mm, rotated rx -180 ry 0 rz 160 deg; joints [14.46, 64.118, -1.835, -142.217, 67.451, 163.444]
  Set speed (17.9 mm/s)
  Call Extruder(1407.66822)
  MoveL 4745 to (480.73, 561.88, 84) mm, rotated rx 180 ry 0 rz 160 deg; joints [14.454, 63.935, -1.431, -142.279, 67.623, 163.592]
  Set speed (17.9 mm/s)
  Call Extruder(1412.00383)
  MoveL 4746 to (479.42, 561.46, 84) mm, rotated rx 180 ry 0 rz 160 deg; joints [14.443, 63.741, -1.002, -142.349, 67.805, 163.752]
  Set speed (17.9 mm/s)
  Call Extruder(1416.23142)
  MoveL 4747 to (478.15, 561.03, 84) mm, rotated rx 180 ry 0 rz 160 deg; joints [14.43, 63.552, -0.586, -142.419, 67.982, 163.907]
  Set speed (17.9 mm/s)
  Call Extruder(1420.41160)
  MoveL 4748 to (476.92, 560.56, 84) mm, rotated rx 180 ry 0 rz 160 deg; joints [14.412, 63.368, -0.178, -142.493, 68.154, 164.061]
  Set speed (17.9 mm/s)
  Call Extruder(1424.55957)
  MoveL 4749 to (475.69, 560.09, 84) mm, rotated rx 180 ry 0 rz 160 deg; joints [14.391, 63.186, 0.224, -142.568, 68.324, 164.213]
  Set speed (17.9 mm/s)
  Call Extruder(1431.94342)
  MoveL 4750 to (473.54, 559.17, 84) mm, rotated rx -180 ry 0 rz 160 deg; joints [14.345, 62.867, 0.933, -142.709, 68.621, 164.485]
  Call Extruder(1437.08641)
  MoveL 4751 to (472.06, 558.49, 84) mm, rotated rx 180 ry 0 rz 160 deg; joints [14.306, 62.648, 1.42, -142.812, 68.825, 164.674]
  Set speed (17.9 mm/s)
  Call Extruder(1441.24137)
  MoveL 4752 to (470.88, 557.91, 84) mm, rotated rx 180 ry 0 rz 160 deg; joints [14.27, 62.473, 1.811, -142.9, 68.987, 164.827]
  Set speed (17.9 mm/s)
  Call Extruder(1444.37304)
  MoveL 4753 to (470, 557.46, 84) mm, rotated rx 180 ry 0 rz 160 deg; joints [14.241, 62.343, 2.103, -142.967, 69.109, 164.942]
  Call Extruder(1450.04423)
  MoveL 4754 to (468.42, 556.61, 84) mm, rotated rx 180 ry 0 rz 160 deg; joints [14.183, 62.109, 2.627, -143.093, 69.325, 165.15]
  Set speed (17.9 mm/s)
  Call Extruder(1453.83840)
  MoveL 4755 to (467.38, 556.01, 84) mm, rotated rx 180 ry 0 rz 160 deg; joints [14.14, 61.954, 2.974, -143.181, 69.468, 165.289]
  Set speed (17.9 mm/s)
  Call Extruder(1457.99625)
  MoveL 4756 to (466.24, 555.33, 84) mm, rotated rx 180 ry 0 rz 160 deg; joints [14.089, 61.787, 3.35, -143.28, 69.623, 165.44]
  Call Extruder(1462.14441)
  MoveL 4757 to (465.13, 554.64, 84) mm, rotated rx -180 ry 0 rz 160 deg; joints [14.035, 61.622, 3.722, -143.382, 69.775, 165.591]
  Set speed (17.9 mm/s)
  Call Extruder(1466.49117)
  MoveL 4758 to (463.97, 553.88, 84) mm, rotated rx 180 ry 0 rz 160 deg; joints [13.974, 61.451, 4.107, -143.491, 69.932, 165.749]
  Call Extruder(1470.55464)
  MoveL 4759 to (462.91, 553.16, 84) mm, rotated rx 180 ry 0 rz 160 deg; joints [13.914, 61.293, 4.463, -143.597, 70.076, 165.895]
  Set speed (17.9 mm/s)
  Call Extruder(1474.73280)
  MoveL 4760 to (461.83, 552.39, 84) mm, rotated rx 180 ry 0 rz 160 deg; joints [13.848, 61.134, 4.824, -143.708, 70.223, 166.046]
  Set speed (17.9 mm/s)
  Call Extruder(1478.89686)
  MoveL 4761 to (460.77, 551.6, 84) mm, rotated rx 180 ry 0 rz 160 deg; joints [13.779, 60.977, 5.18, -143.821, 70.367, 166.195]
  Call Extruder(1483.06850)
  MoveL 4762 to (459.73, 550.78, 84) mm, rotated rx -180 ry 0 rz 160 deg; joints [13.705, 60.822, 5.531, -143.939, 70.508, 166.343]
  Set speed (17.9 mm/s)
  Call Extruder(1487.26777)
  MoveL 4763 to (458.69, 549.95, 84) mm, rotated rx -180 ry 0 rz 160 deg; joints [13.627, 60.668, 5.881, -144.059, 70.648, 166.492]
  Set speed (17.9 mm/s)
  Call Extruder(1491.44042)
  MoveL 4764 to (457.68, 549.09, 84) mm, rotated rx -180 ry 0 rz 160 deg; joints [13.546, 60.518, 6.223, -144.182, 70.785, 166.638]
  Set speed (17.9 mm/s)
  Call Extruder(1495.64288)
  MoveL 4765 to (456.68, 548.21, 84) mm, rotated rx -180 ry 0 rz 160 deg; joints [13.461, 60.369, 6.562, -144.309, 70.92, 166.785]
  Set speed (17.9 mm/s)
  Call Extruder(1499.89722)
  MoveL 4766 to (455.68, 547.3, 84) mm, rotated rx 180 ry 0 rz 160 deg; joints [13.371, 60.221, 6.901, -144.439, 71.054, 166.933]
  Call Extruder(1503.97881)
  MoveL 4767 to (454.75, 546.41, 84) mm, rotated rx -180 ry 0 rz 160 deg; joints [13.281, 60.082, 7.22, -144.568, 71.181, 167.073]
  Set speed (17.9 mm/s)
  Call Extruder(1508.17512)
  MoveL 4768 to (453.81, 545.47, 84) mm, rotated rx 180 ry 0 rz 160 deg; joints [13.184, 59.941, 7.543, -144.703, 71.308, 167.217]
  Call Extruder(1512.32314)
  MoveL 4769 to (452.89, 544.52, 84) mm, rotated rx 180 ry 0 rz 160 deg; joints [13.085, 59.804, 7.857, -144.84, 71.431, 167.357]
  Set speed (17.9 mm/s)
  Call Extruder(1516.52171)
  MoveL 4770 to (451.99, 543.55, 84) mm, rotated rx 180 ry 0 rz 160 deg; joints [12.982, 59.669, 8.169, -144.98, 71.553, 167.498]
  Call Extruder(1520.68493)
  MoveL 4771 to (451.11, 542.56, 84) mm, rotated rx 180 ry 0 rz 160 deg; joints [12.875, 59.537, 8.473, -145.123, 71.67, 167.636]
  Set speed (17.9 mm/s)
  Call Extruder(1524.44633)
  MoveL 4772 to (450.34, 541.65, 84) mm, rotated rx 180 ry 0 rz 160 deg; joints [12.775, 59.42, 8.742, -145.254, 71.775, 167.76]
  Set speed (17.9 mm/s)
  Call Extruder(1529.09855)
  MoveL 4773 to (449.4, 540.51, 84) mm, rotated rx -180 ry 0 rz 160 deg; joints [12.648, 59.279, 9.068, -145.419, 71.9, 167.912]
  Set speed (17.9 mm/s)
  Call Extruder(1533.26828)
  MoveL 4774 to (448.59, 539.47, 84) mm, rotated rx 180 ry 0 rz 160 deg; joints [12.531, 59.156, 9.355, -145.57, 72.01, 168.046]
  Set speed (17.9 mm/s)
  Call Extruder(1537.44319)
  MoveL 4775 to (447.79, 538.42, 84) mm, rotated rx 180 ry 0 rz 160 deg; joints [12.41, 59.035, 9.635, -145.724, 72.117, 168.179]
  Set speed (17.9 mm/s)
  Call Extruder(1541.59102)
  MoveL 4776 to (447.03, 537.35, 84) mm, rotated rx 180 ry 0 rz 160 deg; joints [12.286, 58.918, 9.908, -145.88, 72.22, 168.31]
  Set speed (17.9 mm/s)
  Call Extruder(1545.80523)
  MoveL 4777 to (446.27, 536.25, 84) mm, rotated rx 180 ry 0 rz 160 deg; joints [12.157, 58.801, 10.178, -146.04, 72.322, 168.441]
  Call Extruder(1549.99966)
  MoveL 4778 to (445.54, 535.14, 84) mm, rotated rx 180 ry 0 rz 160 deg; joints [12.024, 58.689, 10.441, -146.203, 72.42, 168.57]
  Set speed (17.9 mm/s)
  Call Extruder(1554.18213)
  MoveL 4779 to (444.83, 534.02, 84) mm, rotated rx 180 ry 0 rz 160 deg; joints [11.889, 58.58, 10.696, -146.367, 72.515, 168.697]
  Set speed (17.9 mm/s)
  Call Extruder(1558.30618)
  MoveL 4780 to (444.15, 532.9, 84) mm, rotated rx 180 ry 0 rz 160 deg; joints [11.753, 58.475, 10.942, -146.532, 72.605, 168.82]
  Set speed (17.9 mm/s)
  Call Extruder(1562.61602)
  MoveL 4781 to (443.47, 531.71, 84) mm, rotated rx 180 ry 0 rz 160 deg; joints [11.607, 58.368, 11.19, -146.706, 72.696, 168.947]
  Set speed (17.9 mm/s)
  Call Extruder(1566.69222)
  MoveL 4782 to (442.85, 530.58, 84) mm, rotated rx 180 ry 0 rz 160 deg; joints [11.466, 58.271, 11.419, -146.873, 72.779, 169.066]
  Set speed (17.9 mm/s)
  Call Extruder(1570.84023)
  MoveL 4783 to (442.24, 529.42, 84) mm, rotated rx 180 ry 0 rz 160 deg; joints [11.32, 58.174, 11.646, -147.046, 72.86, 169.184]
  Call Extruder(0.00000)
  Set speed (17.9 mm/s)
  Call Extruder(4.27937)
  MoveL 4784 to (441.64, 528.2, 84) mm, rotated rx 180 ry 0 rz 160 deg; joints [11.165, 58.078, 11.872, -147.226, 72.941, 169.305]
  Set speed (17.9 mm/s)
  Call Extruder(8.52207)
  MoveL 4785 to (441.07, 526.98, 84) mm, rotated rx 180 ry 0 rz 160 deg; joints [11.009, 57.987, 12.087, -147.407, 73.016, 169.422]
  Set speed (17.9 mm/s)
  Call Extruder(12.52148)
  MoveL 4786 to (440.55, 525.83, 84) mm, rotated rx -180 ry 0 rz 160 deg; joints [10.86, 57.902, 12.286, -147.579, 73.086, 169.531]
  Set speed (17.9 mm/s)
  Call Extruder(16.90057)
  MoveL 4787 to (440.02, 524.55, 84) mm, rotated rx 180 ry 0 rz 160 deg; joints [10.693, 57.815, 12.493, -147.771, 73.156, 169.647]
  Set speed (17.9 mm/s)
  Call Extruder(20.88475)
  MoveL 4788 to (439.55, 523.38, 84) mm, rotated rx 180 ry 0 rz 160 deg; joints [10.539, 57.737, 12.677, -147.946, 73.219, 169.752]
  Set speed (17.9 mm/s)
  Call Extruder(24.76138)
  MoveL 4789 to (439.12, 522.23, 84) mm, rotated rx -180 ry 0 rz 160 deg; joints [10.386, 57.665, 12.847, -148.118, 73.275, 169.852]
  Set speed (17.9 mm/s)
  Call Extruder(29.32342)
  MoveL 4790 to (438.63, 520.87, 84) mm, rotated rx -180 ry 0 rz 160 deg; joints [10.204, 57.583, 13.042, -148.323, 73.339, 169.967]
  Set speed (17.9 mm/s)
  Call Extruder(33.64698)
  MoveL 4791 to (438.21, 519.57, 84) mm, rotated rx 180 ry 0 rz 160 deg; joints [10.028, 57.51, 13.216, -148.519, 73.394, 170.074]
  Set speed (17.9 mm/s)
  Call Extruder(37.73329)
  MoveL 4792 to (437.83, 518.33, 84) mm, rotated rx 180 ry 0 rz 160 deg; joints [9.861, 57.443, 13.375, -148.706, 73.444, 170.173]
  Set speed (17.9 mm/s)
  Call Extruder(42.01827)
  MoveL 4793 to (437.47, 517.02, 84) mm, rotated rx -180 ry 0 rz 160 deg; joints [9.682, 57.377, 13.531, -148.904, 73.491, 170.274]
  Set speed (17.9 mm/s)
  Call Extruder(46.06332)
  MoveL 4794 to (437.14, 515.79, 84) mm, rotated rx 180 ry 0 rz 160 deg; joints [9.512, 57.317, 13.673, -149.091, 73.533, 170.368]
  Set speed (17.9 mm/s)
  Call Extruder(49.79926)
  MoveL 4795 to (436.86, 514.64, 84) mm, rotated rx 180 ry 0 rz 160 deg; joints [9.352, 57.266, 13.796, -149.266, 73.568, 170.453]
  Set speed (17.8 mm/s)
  Call Extruder(55.18161)
  MoveL 4796 to (436.49, 512.98, 84) mm, rotated rx -180 ry 0 rz 160 deg; joints [9.121, 57.195, 13.965, -149.519, 73.614, 170.572]
  Set speed (17.9 mm/s)
  Call Extruder(62.98560)
  MoveL 4797 to (436.05, 510.55, 84) mm, rotated rx -180 ry 0 rz 160 deg; joints [8.779, 57.103, 14.184, -149.89, 73.668, 170.738]
  Set speed (17.9 mm/s)
  Call Extruder(71.35599)
  MoveL 4798 to (435.67, 507.92, 84) mm, rotated rx -180 ry 0 rz 160 deg; joints [8.405, 57.018, 14.388, -150.291, 73.712, 170.908]
  Set speed (17.9 mm/s)
  Call Extruder(79.72425)
  MoveL 4799 to (435.4, 505.28, 84) mm, rotated rx 180 ry 0 rz 160 deg; joints [8.026, 56.946, 14.56, -150.696, 73.739, 171.068]
  Set speed (17.9 mm/s)
  Call Extruder(87.93832)
  MoveL 4800 to (435.24, 502.68, 84) mm, rotated rx -180 ry 0 rz 160 deg; joints [7.649, 56.889, 14.696, -151.095, 73.75, 171.217]
  Set speed (17.9 mm/s)
  Call Extruder(96.37095)
  MoveL 4801 to (435.18, 500.01, 84) mm, rotated rx -180 ry 0 rz 160 deg; joints [7.259, 56.845, 14.802, -151.505, 73.746, 171.361]
  Set speed (17.9 mm/s)
  Call Extruder(103.98555)
  MoveL 4802 to (435.23, 497.6, 84) mm, rotated rx -180 ry 0 rz 160 deg; joints [6.904, 56.817, 14.87, -151.876, 73.728, 171.482]
  Set speed (17.9 mm/s)
  Call Extruder(111.42576)
  MoveL 4803 to (435.36, 495.25, 84) mm, rotated rx -180 ry 0 rz 160 deg; joints [6.556, 56.801, 14.909, -152.238, 73.696, 171.594]
  Call Extruder(118.89226)
  MoveL 4804 to (435.58, 492.89, 84) mm, rotated rx -180 ry 0 rz 160 deg; joints [6.206, 56.795, 14.921, -152.6, 73.652, 171.699]
  Set speed (17.9 mm/s)
  Call Extruder(126.40076)
  MoveL 4805 to (435.88, 490.53, 84) mm, rotated rx 180 ry 0 rz 160 deg; joints [5.854, 56.802, 14.906, -152.962, 73.593, 171.797]
  Call Extruder(134.09938)
  MoveL 4806 to (436.28, 488.12, 84) mm, rotated rx 180 ry 0 rz 160 deg; joints [5.493, 56.819, 14.864, -153.33, 73.52, 171.891]
  Call Extruder(141.48457)
  MoveL 4807 to (436.75, 485.83, 84) mm, rotated rx -180 ry 0 rz 160 deg; joints [5.149, 56.848, 14.796, -153.681, 73.437, 171.973]
  Set speed (17.9 mm/s)
  Call Extruder(149.06901)
  MoveL 4808 to (437.32, 483.49, 84) mm, rotated rx 180 ry 0 rz 160 deg; joints [4.798, 56.888, 14.699, -154.036, 73.337, 172.051]
  Call Extruder(156.51238)
  MoveL 4809 to (437.96, 481.22, 84) mm, rotated rx 180 ry 0 rz 160 deg; joints [4.457, 56.939, 14.577, -154.38, 73.226, 172.121]
  Set speed (17.9 mm/s)
  Call Extruder(164.06072)
  MoveL 4810 to (438.7, 478.95, 84) mm, rotated rx -180 ry 0 rz 160 deg; joints [4.114, 57.001, 14.428, -154.723, 73.101, 172.184]
  Set speed (17.9 mm/s)
  Call Extruder(171.57602)
  MoveL 4811 to (439.51, 476.71, 84) mm, rotated rx 180 ry 0 rz 160 deg; joints [3.777, 57.075, 14.252, -155.059, 72.963, 172.241]
  Set speed (17.9 mm/s)
  Call Extruder(179.26199)
  MoveL 4812 to (440.43, 474.45, 84) mm, rotated rx 180 ry 0 rz 160 deg; joints [3.438, 57.161, 14.045, -155.395, 72.808, 172.292]
  Set speed (17.9 mm/s)
  Call Extruder(186.71543)
  MoveL 4813 to (441.4, 472.3, 84) mm, rotated rx -180 ry 0 rz 160 deg; joints [3.114, 57.256, 13.819, -155.714, 72.645, 172.334]
  Set speed (17.9 mm/s)
  Call Extruder(194.33502)
  MoveL 4814 to (442.48, 470.13, 84) mm, rotated rx -180 ry 0 rz 160 deg; joints [2.79, 57.364, 13.561, -156.032, 72.465, 172.371]
  Set speed (17.9 mm/s)
  Call Extruder(201.76816)
  MoveL 4815 to (443.6, 468.06, 84) mm, rotated rx 180 ry 0 rz 160 deg; joints [2.481, 57.48, 13.286, -156.333, 72.278, 172.401]
  Set speed (17.9 mm/s)
  Call Extruder(209.38937)
  MoveL 4816 to (444.83, 465.98, 84) mm, rotated rx -180 ry 0 rz 160 deg; joints [2.171, 57.61, 12.977, -156.632, 72.074, 172.425]
  Set speed (17.9 mm/s)
  Call Extruder(216.82158)
  MoveL 4817 to (446.1, 464, 84) mm, rotated rx -180 ry 0 rz 160 deg; joints [1.877, 57.748, 12.652, -156.915, 71.862, 172.442]
  Call Extruder(224.34232)
  MoveL 4818 to (447.46, 462.04, 84) mm, rotated rx 180 ry 0 rz 160 deg; joints [1.588, 57.897, 12.3, -157.191, 71.637, 172.453]
  Set speed (17.9 mm/s)
  Call Extruder(231.95522)
  MoveL 4819 to (448.91, 460.11, 84) mm, rotated rx 180 ry 0 rz 160 deg; joints [1.305, 58.059, 11.918, -157.458, 71.397, 172.457]
  Set speed (17.9 mm/s)
  Call Extruder(239.35115)
  MoveL 4820 to (450.39, 458.29, 84) mm, rotated rx -180 ry 0 rz 160 deg; joints [1.039, 58.226, 11.524, -157.707, 71.153, 172.456]
  Set speed (17.9 mm/s)
  Call Extruder(246.93235)
  MoveL 4821 to (451.97, 456.48, 84) mm, rotated rx -180 ry 0 rz 160 deg; joints [0.776, 58.407, 11.099, -157.951, 70.893, 172.448]
  Set speed (17.9 mm/s)
  Call Extruder(254.54536)
  MoveL 4822 to (453.62, 454.72, 84) mm, rotated rx 180 ry 0 rz 160 deg; joints [0.523, 58.599, 10.65, -158.183, 70.621, 172.434]
  Call Extruder(261.97634)
  MoveL 4823 to (455.29, 453.07, 84) mm, rotated rx -180 ry 0 rz 160 deg; joints [0.287, 58.797, 10.19, -158.397, 70.345, 172.413]
  Set speed (17.9 mm/s)
  Call Extruder(269.50920)
  MoveL 4824 to (457.05, 451.45, 84) mm, rotated rx 180 ry 0 rz 160 deg; joints [0.058, 59.006, 9.702, -158.602, 70.056, 172.387]
  Set speed (17.9 mm/s)
  Call Extruder(277.12482)
  MoveL 4825 to (458.89, 449.89, 84) mm, rotated rx 180 ry 0 rz 160 deg; joints [-0.162, 59.228, 9.188, -158.795, 69.755, 172.354]
  Set speed (17.9 mm/s)
  Call Extruder(284.56257)
  MoveL 4826 to (460.74, 448.43, 84) mm, rotated rx -180 ry 0 rz 160 deg; joints [-0.366, 59.453, 8.667, -158.971, 69.452, 172.315]
  Set speed (17.9 mm/s)
  Call Extruder(292.10854)
  MoveL 4827 to (462.67, 447.01, 84) mm, rotated rx 180 ry 0 rz 160 deg; joints [-0.56, 59.691, 8.119, -159.135, 69.136, 172.269]
  Call Extruder(299.51605)
  MoveL 4828 to (464.61, 445.7, 84) mm, rotated rx -180 ry 0 rz 160 deg; joints [-0.74, 59.932, 7.563, -159.283, 68.818, 172.218]
  Set speed (17.9 mm/s)
  Call Extruder(307.24670)
  MoveL 4829 to (466.69, 444.4, 84) mm, rotated rx 180 ry 0 rz 160 deg; joints [-0.915, 60.193, 6.965, -159.422, 68.478, 172.158]
  Set speed (17.9 mm/s)
  Call Extruder(314.77913)
  MoveL 4830 to (468.76, 443.21, 84) mm, rotated rx -180 ry 0 rz 160 deg; joints [-1.073, 60.456, 6.365, -159.544, 68.141, 172.093]
  Set speed (17.9 mm/s)
  Call Extruder(322.30172)
  MoveL 4831 to (470.87, 442.1, 84) mm, rotated rx 180 ry 0 rz 160 deg; joints [-1.219, 60.726, 5.749, -159.651, 67.797, 172.022]
  Set speed (17.9 mm/s)
  Call Extruder(329.75576)
  MoveL 4832 to (473, 441.08, 84) mm, rotated rx 180 ry 0 rz 160 deg; joints [-1.352, 61.002, 5.123, -159.743, 67.45, 171.944]
  Call Extruder(337.36756)
  MoveL 4833 to (475.21, 440.11, 84) mm, rotated rx -180 ry 0 rz 160 deg; joints [-1.475, 61.291, 4.469, -159.822, 67.089, 171.859]
  Set speed (17.9 mm/s)
  Call Extruder(344.73126)
  MoveL 4834 to (477.38, 439.26, 84) mm, rotated rx -180 ry 0 rz 160 deg; joints [-1.582, 61.577, 3.822, -159.885, 66.736, 171.769]
  Set speed (17.9 mm/s)
  Call Extruder(352.38258)
  MoveL 4835 to (479.67, 438.45, 84) mm, rotated rx 180 ry 0 rz 160 deg; joints [-1.681, 61.882, 3.136, -159.935, 66.363, 171.669]
  Call Extruder(359.86889)
  MoveL 4836 to (481.93, 437.75, 84) mm, rotated rx 180 ry 0 rz 160 deg; joints [-1.765, 62.187, 2.451, -159.969, 65.995, 171.563]
  Set speed (17.9 mm/s)
  Call Extruder(367.40026)
  MoveL 4837 to (484.24, 437.13, 84) mm, rotated rx -180 ry 0 rz 160 deg; joints [-1.838, 62.5, 1.751, -159.988, 65.62, 171.45]
  Call Extruder(375.01261)
  MoveL 4838 to (486.59, 436.59, 84) mm, rotated rx 180 ry 0 rz 160 deg; joints [-1.9, 62.823, 1.031, -159.993, 65.238, 171.329]
  Set speed (17.9 mm/s)
  Call Extruder(382.39932)
  MoveL 4839 to (488.89, 436.14, 84) mm, rotated rx -180 ry 0 rz 160 deg; joints [-1.947, 63.142, 0.322, -159.983, 64.864, 171.203]
  Set speed (17.9 mm/s)
  Call Extruder(389.65626)
  MoveL 4840 to (491.16, 435.79, 84) mm, rotated rx 180 ry 0 rz 160 deg; joints [-1.984, 63.46, -0.383, -159.959, 64.495, 171.074]
  Set speed (17.9 mm/s)
  Call Extruder(397.38469)
  MoveL 4841 to (493.59, 435.5, 84) mm, rotated rx 180 ry 0 rz 160 deg; joints [-2.01, 63.804, -1.143, -159.92, 64.1, 170.928]
  Set speed (17.9 mm/s)
  Call Extruder(405.04466)
  MoveL 4842 to (496.01, 435.31, 84) mm, rotated rx 180 ry 0 rz 160 deg; joints [-2.024, 64.15, -1.905, -159.865, 63.707, 170.775]
  Call Extruder(412.66184)
  MoveL 4843 to (498.42, 435.2, 84) mm, rotated rx 180 ry 0 rz 160 deg; joints [-2.026, 64.499, -2.671, -159.796, 63.316, 170.616]
  Set speed (17.9 mm/s)
  Call Extruder(420.11932)
  MoveL 4844 to (500.79, 435.19, 84) mm, rotated rx -180 ry 0 rz 160 deg; joints [-2.018, 64.844, -3.427, -159.714, 62.931, 170.452]
  Set speed (17.9 mm/s)
  Call Extruder(427.54688)
  MoveL 4845 to (503.14, 435.26, 84) mm, rotated rx 180 ry 0 rz 160 deg; joints [-1.998, 65.192, -4.186, -159.619, 62.549, 170.281]
  Call Extruder(435.17426)
  MoveL 4846 to (505.55, 435.42, 84) mm, rotated rx -180 ry 0 rz 160 deg; joints [-1.967, 65.552, -4.97, -159.507, 62.157, 170.098]
  Set speed (17.9 mm/s)
  Call Extruder(442.78048)
  MoveL 4847 to (507.95, 435.67, 84) mm, rotated rx 180 ry 0 rz 160 deg; joints [-1.925, 65.914, -5.756, -159.381, 61.767, 169.908]
  Set speed (17.9 mm/s)
  Call Extruder(450.15718)
  MoveL 4848 to (510.26, 436, 84) mm, rotated rx 180 ry 0 rz 160 deg; joints [-1.875, 66.267, -6.521, -159.246, 61.391, 169.715]
  Call Extruder(457.62041)
  MoveL 4849 to (512.59, 436.42, 84) mm, rotated rx 180 ry 0 rz 160 deg; joints [-1.813, 66.627, -7.298, -159.095, 61.012, 169.513]
  Set speed (17.9 mm/s)
  Call Extruder(464.70476)
  MoveL 4850 to (514.79, 436.89, 84) mm, rotated rx -180 ry 0 rz 160 deg; joints [-1.747, 66.97, -8.036, -158.941, 60.655, 169.314]
  Set speed (17.9 mm/s)
  Call Extruder(472.75916)
  MoveL 4851 to (517.26, 437.52, 84) mm, rotated rx 180 ry 0 rz 160 deg; joints [-1.66, 67.361, -8.876, -158.751, 60.253, 169.08]
  Set speed (17.9 mm/s)
  Call Extruder(480.34498)
  MoveL 4852 to (519.57, 438.21, 84) mm, rotated rx -180 ry 0 rz 160 deg; joints [-1.568, 67.73, -9.668, -158.559, 59.877, 168.851]
  Set speed (17.9 mm/s)
  Call Extruder(487.94587)
  MoveL 4853 to (521.85, 438.98, 84) mm, rotated rx -180 ry 0 rz 160 deg; joints [-1.467, 68.101, -10.459, -158.354, 59.505, 168.613]
  Set speed (17.9 mm/s)
  Call Extruder(495.38843)
  MoveL 4854 to (524.05, 439.81, 84) mm, rotated rx -180 ry 0 rz 160 deg; joints [-1.359, 68.463, -11.232, -158.141, 59.145, 168.374]
  Call Extruder(503.00425)
  MoveL 4855 to (526.28, 440.75, 84) mm, rotated rx 180 ry 0 rz 160 deg; joints [-1.24, 68.833, -12.02, -157.91, 58.782, 168.121]
  Call Extruder(510.53490)
  MoveL 4856 to (528.44, 441.76, 84) mm, rotated rx 180 ry 0 rz 160 deg; joints [-1.114, 69.198, -12.795, -157.671, 58.43, 167.864]
  Set speed (17.9 mm/s)
  Call Extruder(517.98122)
  MoveL 4857 to (530.54, 442.83, 84) mm, rotated rx -180 ry 0 rz 160 deg; joints [-0.98, 69.557, -13.555, -157.423, 58.087, 167.604]
  Set speed (17.9 mm/s)
  Call Extruder(525.57860)
  MoveL 4858 to (532.65, 444, 84) mm, rotated rx -180 ry 0 rz 160 deg; joints [-0.837, 69.922, -14.325, -157.16, 57.744, 167.331]
  Set speed (17.9 mm/s)
  Call Extruder(533.22458)
  MoveL 4859 to (534.72, 445.27, 84) mm, rotated rx 180 ry 0 rz 160 deg; joints [-0.684, 70.286, -15.093, -156.883, 57.406, 167.05]
  Set speed (17.9 mm/s)
  Call Extruder(540.63829)
  MoveL 4860 to (536.68, 446.56, 84) mm, rotated rx 180 ry 0 rz 160 deg; joints [-0.528, 70.636, -15.829, -156.604, 57.087, 166.771]
  Set speed (17.9 mm/s)
  Call Extruder(548.00727)
  MoveL 4861 to (538.58, 447.92, 84) mm, rotated rx 180 ry 0 rz 160 deg; joints [-0.367, 70.98, -16.551, -156.319, 56.777, 166.488]
  Set speed (17.9 mm/s)
  Call Extruder(555.60086)
  MoveL 4862 to (540.49, 449.39, 84) mm, rotated rx 180 ry 0 rz 160 deg; joints [-0.194, 71.33, -17.285, -156.015, 56.467, 166.192]
  Set speed (17.9 mm/s)
  Call Extruder(563.01466)
  MoveL 4863 to (542.3, 450.89, 84) mm, rotated rx 180 ry 0 rz 160 deg; joints [-0.018, 71.668, -17.99, -155.71, 56.174, 165.897]
  Set speed (17.9 mm/s)
  Call Extruder(570.74211)
  MoveL 4864 to (544.13, 452.52, 84) mm, rotated rx -180 ry 0 rz 160 deg; joints [0.172, 72.014, -18.713, -155.383, 55.878, 165.585]
  Set speed (17.9 mm/s)
  Call Extruder(578.21298)
  MoveL 4865 to (545.83, 454.17, 84) mm, rotated rx 180 ry 0 rz 160 deg; joints [0.362, 72.342, -19.398, -155.059, 55.602, 165.28]
  Set speed (17.9 mm/s)
  Call Extruder(582.35094)
  MoveL 4866 to (546.75, 455.1, 84) mm, rotated rx -180 ry 0 rz 160 deg; joints [0.469, 72.521, -19.77, -154.877, 55.455, 165.109]
  Set speed (17.9 mm/s)
  Call Extruder(586.47658)
  MoveL 4867 to (547.65, 456.06, 84) mm, rotated rx 180 ry 0 rz 160 deg; joints [0.578, 72.698, -20.136, -154.693, 55.311, 164.938]
  Set speed (17.9 mm/s)
  Call Extruder(590.69148)
  MoveL 4868 to (548.54, 457.05, 84) mm, rotated rx -180 ry 0 rz 160 deg; joints [0.691, 72.876, -20.507, -154.503, 55.167, 164.762]
  Set speed (17.9 mm/s)
  Call Extruder(594.83044)
  MoveL 4869 to (549.4, 458.04, 84) mm, rotated rx 180 ry 0 rz 160 deg; joints [0.804, 73.048, -20.864, -154.315, 55.03, 164.589]
  Call Extruder(599.00428)
  MoveL 4870 to (550.25, 459.06, 84) mm, rotated rx 180 ry 0 rz 160 deg; joints [0.919, 73.22, -21.22, -154.123, 54.895, 164.413]
  Set speed (17.9 mm/s)
  Call Extruder(603.23761)
  MoveL 4871 to (551.09, 460.11, 84) mm, rotated rx 180 ry 0 rz 160 deg; joints [1.038, 73.391, -21.575, -153.926, 54.762, 164.234]
  Call Extruder(607.36902)
  MoveL 4872 to (551.88, 461.15, 84) mm, rotated rx -180 ry 0 rz 160 deg; joints [1.155, 73.556, -21.915, -153.733, 54.636, 164.059]
  Set speed (17.9 mm/s)
  Call Extruder(611.01554)
  MoveL 4873 to (552.57, 462.08, 84) mm, rotated rx 180 ry 0 rz 160 deg; joints [1.26, 73.699, -22.211, -153.562, 54.528, 163.904]
  Set speed (17.9 mm/s)
  Call Extruder(615.71639)
  MoveL 4874 to (553.42, 463.3, 84) mm, rotated rx 180 ry 0 rz 160 deg; joints [1.396, 73.879, -22.584, -153.339, 54.394, 163.705]
  Set speed (17.9 mm/s)
  Call Extruder(619.49806)
  MoveL 4875 to (554.09, 464.29, 84) mm, rotated rx 180 ry 0 rz 160 deg; joints [1.508, 74.022, -22.88, -153.158, 54.289, 163.544]
  Set speed (17.9 mm/s)
  Call Extruder(624.08649)
  MoveL 4876 to (554.88, 465.51, 84) mm, rotated rx -180 ry 0 rz 160 deg; joints [1.644, 74.193, -23.231, -152.938, 54.167, 163.349]
  Set speed (17.9 mm/s)
  Call Extruder(628.34082)
  MoveL 4877 to (555.59, 466.66, 84) mm, rotated rx 180 ry 0 rz 160 deg; joints [1.772, 74.346, -23.548, -152.733, 54.058, 163.168]
  Set speed (17.9 mm/s)
  Call Extruder(632.47216)
  MoveL 4878 to (556.25, 467.79, 84) mm, rotated rx 180 ry 0 rz 160 deg; joints [1.898, 74.492, -23.849, -152.533, 53.957, 162.993]
  Set speed (17.9 mm/s)
  Call Extruder(637.94566)
  MoveL 4879 to (557.09, 469.31, 84) mm, rotated rx 180 ry 0 rz 160 deg; joints [2.066, 74.681, -24.237, -152.266, 53.83, 162.761]
  Set speed (17.9 mm/s)
  Call Extruder(640.96406)
  MoveL 4880 to (557.54, 470.15, 84) mm, rotated rx -180 ry 0 rz 160 deg; joints [2.16, 74.782, -24.445, -152.119, 53.763, 162.634]
  Set speed (17.9 mm/s)
  Call Extruder(645.05491)
  MoveL 4881 to (558.12, 471.31, 84) mm, rotated rx -180 ry 0 rz 160 deg; joints [2.287, 74.917, -24.722, -151.919, 53.676, 162.462]
  Set speed (17.9 mm/s)
  Call Extruder(650.37457)
  MoveL 4882 to (558.85, 472.83, 84) mm, rotated rx 180 ry 0 rz 160 deg; joints [2.455, 75.086, -25.07, -151.658, 53.569, 162.239]
  Set speed (17.9 mm/s)
  Call Extruder(653.45917)
  MoveL 4883 to (559.25, 473.72, 84) mm, rotated rx 180 ry 0 rz 160 deg; joints [2.553, 75.181, -25.264, -151.507, 53.512, 162.111]
  Set speed (17.9 mm/s)
  Call Extruder(657.67880)
  MoveL 4884 to (559.77, 474.95, 84) mm, rotated rx 180 ry 0 rz 160 deg; joints [2.689, 75.307, -25.523, -151.299, 53.437, 161.937]
  Call Extruder(661.86352)
  MoveL 4885 to (560.28, 476.17, 84) mm, rotated rx -180 ry 0 rz 160 deg; joints [2.823, 75.43, -25.775, -151.094, 53.366, 161.764]
  Set speed (17.9 mm/s)
  Call Extruder(666.03788)
  MoveL 4886 to (560.75, 477.41, 84) mm, rotated rx -180 ry 0 rz 160 deg; joints [2.959, 75.546, -26.012, -150.889, 53.302, 161.594]
  Call Extruder(670.18874)
  MoveL 4887 to (561.2, 478.64, 84) mm, rotated rx 180 ry 0 rz 160 deg; joints [3.095, 75.659, -26.244, -150.686, 53.242, 161.426]
  Call Extruder(674.42991)
  MoveL 4888 to (561.62, 479.92, 84) mm, rotated rx 180 ry 0 rz 160 deg; joints [3.235, 75.769, -26.469, -150.478, 53.187, 161.257]
  Call Extruder(678.53050)
  MoveL 4889 to (562.02, 481.15, 84) mm, rotated rx 180 ry 0 rz 160 deg; joints [3.37, 75.872, -26.68, -150.278, 53.136, 161.094]
  Set speed (17.9 mm/s)
  Call Extruder(682.79587)
  MoveL 4890 to (562.39, 482.45, 84) mm, rotated rx -180 ry 0 rz 160 deg; joints [3.512, 75.973, -26.886, -150.07, 53.091, 160.927]
  Call Extruder(686.79937)
  MoveL 4891 to (562.73, 483.67, 84) mm, rotated rx -180 ry 0 rz 160 deg; joints [3.646, 76.065, -27.075, -149.876, 53.052, 160.772]
  Set speed (17.9 mm/s)
  Call Extruder(691.18259)
  MoveL 4892 to (563.06, 485.02, 84) mm, rotated rx 180 ry 0 rz 160 deg; joints [3.794, 76.159, -27.267, -149.664, 53.016, 160.605]
  Call Extruder(695.27897)
  MoveL 4893 to (563.35, 486.28, 84) mm, rotated rx 180 ry 0 rz 160 deg; joints [3.933, 76.244, -27.441, -149.467, 52.985, 160.451]
  Set speed (17.9 mm/s)
  Call Extruder(703.70292)
  MoveL 4894 to (563.86, 488.9, 84) mm, rotated rx 180 ry 0 rz 160 deg; joints [4.22, 76.402, -27.764, -149.064, 52.94, 160.141]
  Call Extruder(712.00042)
  MoveL 4895 to (564.26, 491.5, 84) mm, rotated rx 180 ry 0 rz 160 deg; joints [4.505, 76.538, -28.042, -148.673, 52.917, 159.847]
  Set speed (17.9 mm/s)
  Call Extruder(720.53140)
  MoveL 4896 to (564.55, 494.19, 84) mm, rotated rx -180 ry 0 rz 160 deg; joints [4.8, 76.657, -28.283, -148.278, 52.915, 159.557]
  Set speed (17.9 mm/s)
  Call Extruder(728.80231)
  MoveL 4897 to (564.74, 496.81, 84) mm, rotated rx 180 ry 0 rz 160 deg; joints [5.088, 76.751, -28.475, -147.901, 52.933, 159.289]
  Call Extruder(737.17025)
  MoveL 4898 to (564.82, 499.46, 84) mm, rotated rx -180 ry 0 rz 160 deg; joints [5.38, 76.825, -28.626, -147.528, 52.972, 159.031]
  Set speed (17.9 mm/s)
  Call Extruder(745.74647)
  MoveL 4899 to (564.78, 502.18, 84) mm, rotated rx 180 ry 0 rz 160 deg; joints [5.68, 76.878, -28.733, -147.155, 53.034, 158.783]
  Set speed (17.9 mm/s)
  Call Extruder(753.89679)
  MoveL 4900 to (564.64, 504.76, 84) mm, rotated rx -180 ry 0 rz 160 deg; joints [5.967, 76.907, -28.792, -146.809, 53.113, 158.562]
  Set speed (17.9 mm/s)
  Call Extruder(762.16810)
  MoveL 4901 to (564.4, 507.37, 84) mm, rotated rx -180 ry 0 rz 160 deg; joints [6.257, 76.914, -28.808, -146.468, 53.213, 158.354]
  Call Extruder(770.71650)
  MoveL 4902 to (564.03, 510.05, 84) mm, rotated rx 180 ry 0 rz 160 deg; joints [6.558, 76.9, -28.779, -146.126, 53.336, 158.156]
  Set speed (17.9 mm/s)
  Call Extruder(778.97109)
  MoveL 4903 to (563.58, 512.63, 84) mm, rotated rx -180 ry 0 rz 160 deg; joints [6.847, 76.864, -28.706, -145.806, 53.475, 157.982]
  Set speed (17.9 mm/s)
  Call Extruder(787.40253)
  MoveL 4904 to (563, 515.24, 84) mm, rotated rx -180 ry 0 rz 160 deg; joints [7.143, 76.805, -28.586, -145.492, 53.637, 157.823]
  Set speed (17.9 mm/s)
  Call Extruder(791.55741)
  MoveL 4905 to (562.67, 516.51, 84) mm, rotated rx -180 ry 0 rz 160 deg; joints [7.287, 76.767, -28.508, -145.342, 53.724, 157.753]
  Call Extruder(795.73960)
  MoveL 4906 to (562.33, 517.79, 84) mm, rotated rx -180 ry 0 rz 160 deg; joints [7.433, 76.726, -28.425, -145.192, 53.814, 157.684]
  Set speed (17.9 mm/s)
  Call Extruder(803.98292)
  MoveL 4907 to (561.56, 520.29, 84) mm, rotated rx 180 ry 0 rz 160 deg; joints [7.72, 76.626, -28.221, -144.908, 54.008, 157.565]
  Set speed (17.9 mm/s)
  Call Extruder(808.28967)
  MoveL 4908 to (561.11, 521.58, 84) mm, rotated rx -180 ry 0 rz 160 deg; joints [7.868, 76.565, -28.095, -144.765, 54.118, 157.511]
  Call Extruder(812.60219)
  MoveL 4909 to (560.65, 522.86, 84) mm, rotated rx 180 ry 0 rz 160 deg; joints [8.017, 76.501, -27.965, -144.624, 54.229, 157.459]
  Set speed (17.9 mm/s)
  Call Extruder(816.66054)
  MoveL 4910 to (560.18, 524.06, 84) mm, rotated rx -180 ry 0 rz 160 deg; joints [8.156, 76.432, -27.825, -144.495, 54.34, 157.417]
  Set speed (17.9 mm/s)
  Call Extruder(820.85178)
  MoveL 4911 to (559.68, 525.29, 84) mm, rotated rx 180 ry 0 rz 160 deg; joints [8.299, 76.36, -27.676, -144.364, 54.457, 157.377]
  Call Extruder(825.05130)
  MoveL 4912 to (559.14, 526.5, 84) mm, rotated rx 180 ry 0 rz 160 deg; joints [8.442, 76.279, -27.513, -144.237, 54.58, 157.343]
  Call Extruder(829.04943)
  MoveL 4913 to (558.62, 527.65, 84) mm, rotated rx 180 ry 0 rz 160 deg; joints [8.578, 76.201, -27.352, -144.117, 54.698, 157.313]
  Set speed (17.9 mm/s)
  Call Extruder(832.34023)
  MoveL 4914 to (558.17, 528.59, 84) mm, rotated rx -180 ry 0 rz 160 deg; joints [8.689, 76.132, -27.212, -144.021, 54.799, 157.292]
  Set speed (17.9 mm/s)
  Call Extruder(837.52048)
  MoveL 4915 to (557.43, 530.06, 84) mm, rotated rx -180 ry 0 rz 160 deg; joints [8.863, 76.017, -26.977, -143.875, 54.963, 157.265]
  Set speed (17.9 mm/s)
  Call Extruder(841.71046)
  MoveL 4916 to (556.8, 531.23, 84) mm, rotated rx 180 ry 0 rz 160 deg; joints [9.003, 75.919, -26.777, -143.759, 55.1, 157.248]
  Set speed (17.9 mm/s)
  Call Extruder(845.99336)
  MoveL 4917 to (556.13, 532.41, 84) mm, rotated rx -180 ry 0 rz 160 deg; joints [9.146, 75.814, -26.561, -143.645, 55.244, 157.237]
  Set speed (17.9 mm/s)
  Call Extruder(850.03716)
  MoveL 4918 to (555.48, 533.51, 84) mm, rotated rx -180 ry 0 rz 160 deg; joints [9.279, 75.71, -26.35, -143.539, 55.383, 157.229]
  Call Extruder(854.25325)
  MoveL 4919 to (554.78, 534.65, 84) mm, rotated rx 180 ry 0 rz 160 deg; joints [9.418, 75.598, -26.12, -143.432, 55.531, 157.226]
  Set speed (17.9 mm/s)
  Call Extruder(858.15814)
  MoveL 4920 to (554.11, 535.69, 84) mm, rotated rx -180 ry 0 rz 160 deg; joints [9.545, 75.49, -25.899, -143.336, 55.671, 157.228]
  Set speed (17.9 mm/s)
  Call Extruder(863.31693)
  MoveL 4921 to (553.19, 537.04, 84) mm, rotated rx 180 ry 0 rz 160 deg; joints [9.712, 75.342, -25.594, -143.213, 55.861, 157.236]
  Set speed (17.9 mm/s)
  Call Extruder(866.81094)
  MoveL 4922 to (552.55, 537.95, 84) mm, rotated rx 180 ry 0 rz 160 deg; joints [9.825, 75.238, -25.382, -143.132, 55.992, 157.244]
  Set speed (17.9 mm/s)
  Call Extruder(870.98282)
  MoveL 4923 to (551.76, 539.01, 84) mm, rotated rx 180 ry 0 rz 160 deg; joints [9.958, 75.11, -25.119, -143.039, 56.151, 157.259]
  Call Extruder(875.15617)
  MoveL 4924 to (550.96, 540.06, 84) mm, rotated rx -180 ry 0 rz 160 deg; joints [10.09, 74.979, -24.849, -142.948, 56.313, 157.278]
  Set speed (17.9 mm/s)
  Call Extruder(879.39252)
  MoveL 4925 to (550.12, 541.11, 84) mm, rotated rx -180 ry 0 rz 160 deg; joints [10.223, 74.841, -24.566, -142.859, 56.48, 157.302]
  Set speed (17.9 mm/s)
  Call Extruder(883.54056)
  MoveL 4926 to (549.27, 542.11, 84) mm, rotated rx -180 ry 0 rz 160 deg; joints [10.352, 74.703, -24.282, -142.774, 56.646, 157.329]
  Set speed (17.9 mm/s)
  Call Extruder(887.70372)
  MoveL 4927 to (548.41, 543.11, 84) mm, rotated rx -180 ry 0 rz 160 deg; joints [10.48, 74.56, -23.989, -142.693, 56.815, 157.36]
  Set speed (17.9 mm/s)
  Call Extruder(892.11759)
  MoveL 4928 to (547.46, 544.14, 84) mm, rotated rx -180 ry 0 rz 160 deg; joints [10.615, 74.406, -23.67, -142.609, 56.997, 157.398]
  Set speed (17.9 mm/s)
  Call Extruder(896.09016)
  MoveL 4929 to (546.6, 545.06, 84) mm, rotated rx -180 ry 0 rz 160 deg; joints [10.735, 74.263, -23.376, -142.536, 57.164, 157.436]
  Set speed (17.9 mm/s)
  Call Extruder(900.28375)
  MoveL 4930 to (545.66, 546, 84) mm, rotated rx 180 ry 0 rz 160 deg; joints [10.861, 74.109, -23.059, -142.463, 57.341, 157.479]
  Call Extruder(904.55796)
  MoveL 4931 to (544.69, 546.95, 84) mm, rotated rx 180 ry 0 rz 160 deg; joints [10.987, 73.95, -22.729, -142.39, 57.524, 157.528]
  Set speed (17.9 mm/s)
  Call Extruder(908.61633)
  MoveL 4932 to (543.75, 547.83, 84) mm, rotated rx 180 ry 0 rz 160 deg; joints [11.106, 73.795, -22.41, -142.324, 57.7, 157.577]
  Set speed (17.9 mm/s)
  Call Extruder(912.80651)
  MoveL 4933 to (542.76, 548.71, 84) mm, rotated rx -180 ry 0 rz 160 deg; joints [11.227, 73.632, -22.073, -142.259, 57.884, 157.632]
  Set speed (17.9 mm/s)
  Call Extruder(917.05969)
  MoveL 4934 to (541.74, 549.59, 84) mm, rotated rx 180 ry 0 rz 160 deg; joints [11.348, 73.464, -21.726, -142.195, 58.072, 157.692]
  Set speed (17.9 mm/s)
  Call Extruder(921.17914)
  MoveL 4935 to (540.73, 550.42, 84) mm, rotated rx -180 ry 0 rz 160 deg; joints [11.464, 73.298, -21.383, -142.136, 58.256, 157.753]
  Set speed (17.9 mm/s)
  Call Extruder(925.40854)
  MoveL 4936 to (539.68, 551.25, 84) mm, rotated rx -180 ry 0 rz 160 deg; joints [11.582, 73.126, -21.026, -142.078, 58.446, 157.819]
  Set speed (17.9 mm/s)
  Call Extruder(929.55083)
  MoveL 4937 to (538.64, 552.04, 84) mm, rotated rx -180 ry 0 rz 160 deg; joints [11.695, 72.955, -20.671, -142.024, 58.634, 157.888]
  Set speed (17.9 mm/s)
  Call Extruder(933.74850)
  MoveL 4938 to (537.56, 552.83, 84) mm, rotated rx 180 ry 0 rz 160 deg; joints [11.809, 72.779, -20.305, -141.972, 58.826, 157.96]
  Set speed (17.9 mm/s)
  Call Extruder(937.90427)
  MoveL 4939 to (536.48, 553.58, 84) mm, rotated rx 180 ry 0 rz 160 deg; joints [11.919, 72.602, -19.938, -141.923, 59.017, 158.036]
  Call Extruder(942.13712)
  MoveL 4940 to (535.36, 554.32, 84) mm, rotated rx 180 ry 0 rz 160 deg; joints [12.03, 72.42, -19.559, -141.876, 59.213, 158.116]
  Set speed (17.9 mm/s)
  Call Extruder(946.28158)
  MoveL 4941 to (534.25, 555.03, 84) mm, rotated rx -180 ry 0 rz 160 deg; joints [12.137, 72.239, -19.183, -141.833, 59.407, 158.197]
  Set speed (17.9 mm/s)
  Call Extruder(950.45950)
  MoveL 4942 to (533.12, 555.72, 84) mm, rotated rx -180 ry 0 rz 160 deg; joints [12.242, 72.055, -18.799, -141.791, 59.603, 158.283]
  Set speed (17.9 mm/s)
  Call Extruder(954.64399)
  MoveL 4943 to (531.98, 556.38, 84) mm, rotated rx 180 ry 0 rz 160 deg; joints [12.346, 71.869, -18.412, -141.752, 59.8, 158.371]
  Set speed (17.9 mm/s)
  Call Extruder(958.24792)
  MoveL 4944 to (530.98, 556.94, 84) mm, rotated rx 180 ry 0 rz 160 deg; joints [12.435, 71.708, -18.075, -141.721, 59.97, 158.449]
  Set speed (17.9 mm/s)
  Call Extruder(964.23636)
  MoveL 4945 to (529.3, 557.82, 84) mm, rotated rx 180 ry 0 rz 160 deg; joints [12.577, 71.437, -17.508, -141.673, 60.254, 158.584]
  Set speed (17.9 mm/s)
  Call Extruder(967.24448)
  MoveL 4946 to (528.45, 558.24, 84) mm, rotated rx -180 ry 0 rz 160 deg; joints [12.647, 71.299, -17.22, -141.651, 60.398, 158.654]
  Set speed (17.9 mm/s)
  Call Extruder(971.34601)
  MoveL 4947 to (527.27, 558.8, 84) mm, rotated rx -180 ry 0 rz 160 deg; joints [12.742, 71.11, -16.824, -141.623, 60.594, 158.752]
  Set speed (17.9 mm/s)
  Call Extruder(975.64478)
  MoveL 4948 to (526.03, 559.36, 84) mm, rotated rx 180 ry 0 rz 160 deg; joints [12.837, 70.91, -16.405, -141.597, 60.801, 158.858]
  Set speed (17.9 mm/s)
  Call Extruder(979.82627)
  MoveL 4949 to (524.81, 559.88, 84) mm, rotated rx 180 ry 0 rz 160 deg; joints [12.929, 70.716, -15.997, -141.572, 61.001, 158.962]
  Call Extruder(984.01552)
  MoveL 4950 to (523.58, 560.37, 84) mm, rotated rx -180 ry 0 rz 160 deg; joints [13.018, 70.519, -15.582, -141.552, 61.203, 159.071]
  Set speed (17.9 mm/s)
  Call Extruder(988.02824)
  MoveL 4951 to (522.39, 560.82, 84) mm, rotated rx -180 ry 0 rz 160 deg; joints [13.102, 70.33, -15.185, -141.534, 61.396, 159.175]
  Set speed (17.9 mm/s)
  Call Extruder(992.44095)
  MoveL 4952 to (521.08, 561.29, 84) mm, rotated rx -180 ry 0 rz 160 deg; joints [13.191, 70.12, -14.743, -141.517, 61.61, 159.295]
  Set speed (17.9 mm/s)
  Call Extruder(996.63821)
  MoveL 4953 to (519.82, 561.71, 84) mm, rotated rx -180 ry 0 rz 160 deg; joints [13.275, 69.921, -14.323, -141.503, 61.812, 159.409]
  Set speed (17.9 mm/s)
  Call Extruder(1001.66451)
  MoveL 4954 to (518.3, 562.18, 84) mm, rotated rx 180 ry 0 rz 160 deg; joints [13.37, 69.68, -13.815, -141.49, 62.055, 159.55]
  Set speed (17.9 mm/s)
  Call Extruder(1004.82204)
  MoveL 4955 to (517.34, 562.45, 84) mm, rotated rx 180 ry 0 rz 160 deg; joints [13.429, 69.529, -13.495, -141.484, 62.207, 159.64]
  Set speed (17.9 mm/s)
  Call Extruder(1008.60333)
  MoveL 4956 to (516.18, 562.76, 84) mm, rotated rx -180 ry 0 rz 160 deg; joints [13.497, 69.347, -13.109, -141.478, 62.39, 159.749]
  Set speed (17.9 mm/s)
  Call Extruder(1013.19607)
  MoveL 4957 to (514.77, 563.11, 84) mm, rotated rx 180 ry 0 rz 160 deg; joints [13.577, 69.126, -12.64, -141.473, 62.611, 159.884]
  Set speed (17.9 mm/s)
  Call Extruder(1021.70749)
  MoveL 4958 to (512.13, 563.67, 84) mm, rotated rx -180 ry 0 rz 160 deg; joints [13.717, 68.713, -11.765, -141.473, 63.022, 160.141]
  Set speed (17.9 mm/s)
  Call Extruder(1030.12426)
  MoveL 4959 to (509.5, 564.12, 84) mm, rotated rx 180 ry 0 rz 160 deg; joints [13.846, 68.304, -10.893, -141.483, 63.427, 160.402]
  Set speed (17.9 mm/s)
  Call Extruder(1038.31484)
  MoveL 4960 to (506.93, 564.45, 84) mm, rotated rx 180 ry 0 rz 160 deg; joints [13.96, 67.905, -10.042, -141.503, 63.819, 160.663]
  Set speed (17.9 mm/s)
  Call Extruder(1046.82063)
  MoveL 4961 to (504.24, 564.68, 84) mm, rotated rx -180 ry 0 rz 160 deg; joints [14.067, 67.491, -9.155, -141.534, 64.224, 160.941]
  Set speed (17.9 mm/s)
  Call Extruder(1055.23893)
  MoveL 4962 to (501.57, 564.8, 84) mm, rotated rx 180 ry 0 rz 160 deg; joints [14.161, 67.081, -8.276, -141.575, 64.622, 161.222]
  Set speed (17.9 mm/s)
  Call Extruder(1063.50853)
  MoveL 4963 to (498.95, 564.81, 84) mm, rotated rx -180 ry 0 rz 160 deg; joints [14.241, 66.68, -7.413, -141.626, 65.01, 161.503]
  Set speed (10.0 mm/s)
  MoveL 4964 to (498.95, 564.81, 88) mm, rotated rx -180 ry 0 rz 160 deg; joints [14.241, 66.029, -7.077, -141.533, 64.763, 161.287]
  Set speed (120.0 mm/s)
  MoveL 4965 to (498.97, 565.19, 88) mm, rotated rx 180 ry 0 rz 160 deg; joints [14.286, 66.046, -7.115, -141.48, 64.761, 161.252]
  Set speed (17.9 mm/s)
  Call Extruder(1072.04379)
  MoveL 4966 to (496.26, 565.09, 88) mm, rotated rx 180 ry 0 rz 160 deg; joints [14.358, 65.632, -6.226, -141.544, 65.156, 161.547]
  Set speed (17.9 mm/s)
  Call Extruder(1080.45395)
  MoveL 4967 to (493.59, 564.88, 88) mm, rotated rx 180 ry 0 rz 160 deg; joints [14.415, 65.226, -5.352, -141.617, 65.541, 161.842]
  Set speed (18.0 mm/s)
  Call Extruder(1088.76267)
  MoveL 4968 to (490.97, 564.57, 88) mm, rotated rx 180 ry 0 rz 160 deg; joints [14.46, 64.828, -4.492, -141.7, 65.916, 162.137]
  Set speed (18.0 mm/s)
  Call Extruder(1097.04705)
  MoveL 4969 to (488.36, 564.15, 88) mm, rotated rx -180 ry 0 rz 160 deg; joints [14.491, 64.434, -3.64, -141.794, 66.286, 162.435]
  Set speed (17.9 mm/s)
  Call Extruder(1105.34849)
  MoveL 4970 to (485.78, 563.63, 88) mm, rotated rx -180 ry 0 rz 160 deg; joints [14.509, 64.044, -2.792, -141.898, 66.651, 162.735]
  Set speed (17.9 mm/s)
  Call Extruder(1109.76951)
  MoveL 4971 to (484.41, 563.3, 88) mm, rotated rx -180 ry 0 rz 160 deg; joints [14.512, 63.838, -2.345, -141.958, 66.842, 162.896]
  Call Extruder(1114.05577)
  MoveL 4972 to (483.09, 562.97, 88) mm, rotated rx 180 ry 0 rz 160 deg; joints [14.513, 63.64, -1.913, -142.019, 67.026, 163.052]
  Set speed (17.9 mm/s)
  Call Extruder(1118.11720)
  MoveL 4973 to (481.85, 562.61, 88) mm, rotated rx -180 ry 0 rz 160 deg; joints [14.509, 63.454, -1.506, -142.08, 67.199, 163.201]
  Set speed (17.9 mm/s)
  Call Extruder(1122.17547)
  MoveL 4974 to (480.62, 562.25, 88) mm, rotated rx 180 ry 0 rz 160 deg; joints [14.503, 63.269, -1.102, -142.143, 67.371, 163.35]
  Set speed (17.9 mm/s)
  Call Extruder(1126.52902)
  MoveL 4975 to (479.3, 561.82, 88) mm, rotated rx -180 ry 0 rz 160 deg; joints [14.492, 63.072, -0.67, -142.214, 67.553, 163.51]
  Set speed (17.9 mm/s)
  Call Extruder(1130.76197)
  MoveL 4976 to (478.03, 561.38, 88) mm, rotated rx 180 ry 0 rz 160 deg; joints [14.479, 62.882, -0.253, -142.285, 67.729, 163.665]
  Set speed (17.9 mm/s)
  Call Extruder(1134.97597)
  MoveL 4977 to (476.78, 560.91, 88) mm, rotated rx 180 ry 0 rz 160 deg; joints [14.46, 62.694, 0.159, -142.36, 67.901, 163.821]
  Call Extruder(1139.01032)
  MoveL 4978 to (475.58, 560.45, 88) mm, rotated rx 180 ry 0 rz 160 deg; joints [14.441, 62.516, 0.551, -142.433, 68.065, 163.969]
  Call Extruder(1143.76201)
  MoveL 4979 to (474.19, 559.87, 88) mm, rotated rx -180 ry 0 rz 160 deg; joints [14.412, 62.308, 1.009, -142.524, 68.256, 164.144]
  Set speed (17.9 mm/s)
  Call Extruder(1147.37406)
  MoveL 4980 to (473.14, 559.41, 88) mm, rotated rx 180 ry 0 rz 160 deg; joints [14.388, 62.151, 1.355, -142.594, 68.4, 164.277]
  Set speed (18.0 mm/s)
  Call Extruder(1151.67565)
  MoveL 4981 to (471.9, 558.83, 88) mm, rotated rx -180 ry 0 rz 160 deg; joints [14.355, 61.966, 1.765, -142.682, 68.569, 164.436]
  Set speed (18.0 mm/s)
  Call Extruder(1155.83242)
  MoveL 4982 to (470.71, 558.25, 88) mm, rotated rx -180 ry 0 rz 160 deg; joints [14.319, 61.789, 2.157, -142.77, 68.731, 164.589]
  Set speed (17.9 mm/s)
  Call Extruder(1158.92817)
  MoveL 4983 to (469.84, 557.8, 88) mm, rotated rx -180 ry 0 rz 160 deg; joints [14.291, 61.659, 2.446, -142.837, 68.85, 164.703]
  Set speed (17.9 mm/s)
  Call Extruder(1164.20159)
  MoveL 4984 to (468.36, 557, 88) mm, rotated rx -180 ry 0 rz 160 deg; joints [14.236, 61.439, 2.935, -142.956, 69.05, 164.897]
  Set speed (18.0 mm/s)
  Call Extruder(1168.38446)
  MoveL 4985 to (467.2, 556.35, 88) mm, rotated rx 180 ry 0 rz 160 deg; joints [14.19, 61.267, 3.319, -143.052, 69.206, 165.051]
  Set speed (17.9 mm/s)
  Call Extruder(1172.62344)
  MoveL 4986 to (466.04, 555.66, 88) mm, rotated rx 180 ry 0 rz 160 deg; joints [14.138, 61.094, 3.703, -143.154, 69.363, 165.206]
  Set speed (17.9 mm/s)
  Call Extruder(1176.81374)
  MoveL 4987 to (464.91, 554.95, 88) mm, rotated rx 180 ry 0 rz 160 deg; joints [14.083, 60.926, 4.079, -143.257, 69.515, 165.358]
  Call Extruder(1181.06382)
  MoveL 4988 to (463.78, 554.21, 88) mm, rotated rx 180 ry 0 rz 160 deg; joints [14.024, 60.757, 4.456, -143.365, 69.667, 165.513]
  Set speed (17.9 mm/s)
  Call Extruder(1185.22510)
  MoveL 4989 to (462.69, 553.46, 88) mm, rotated rx -180 ry 0 rz 160 deg; joints [13.961, 60.594, 4.821, -143.474, 69.814, 165.663]
  Call Extruder(1189.35489)
  MoveL 4990 to (461.62, 552.7, 88) mm, rotated rx -180 ry 0 rz 160 deg; joints [13.896, 60.435, 5.179, -143.584, 69.958, 165.812]
  Set speed (18.0 mm/s)
  Call Extruder(1193.57819)
  MoveL 4991 to (460.54, 551.9, 88) mm, rotated rx -180 ry 0 rz 160 deg; joints [13.826, 60.274, 5.541, -143.7, 70.102, 165.964]
  Set speed (17.9 mm/s)
  Call Extruder(1197.75007)
  MoveL 4992 to (459.49, 551.09, 88) mm, rotated rx 180 ry 0 rz 160 deg; joints [13.752, 60.117, 5.893, -143.818, 70.243, 166.112]
  Set speed (17.9 mm/s)
  Call Extruder(1201.97236)
  MoveL 4993 to (458.45, 550.24, 88) mm, rotated rx -180 ry 0 rz 160 deg; joints [13.674, 59.961, 6.245, -143.94, 70.382, 166.262]
  Set speed (17.9 mm/s)
  Call Extruder(1206.17373)
  MoveL 4994 to (457.43, 549.38, 88) mm, rotated rx 180 ry 0 rz 160 deg; joints [13.592, 59.809, 6.59, -144.064, 70.518, 166.41]
  Call Extruder(1210.36950)
  MoveL 4995 to (456.43, 548.5, 88) mm, rotated rx -180 ry 0 rz 160 deg; joints [13.507, 59.658, 6.93, -144.191, 70.652, 166.557]
  Set speed (17.9 mm/s)
  Call Extruder(1214.51873)
  MoveL 4996 to (455.45, 547.61, 88) mm, rotated rx -180 ry 0 rz 160 deg; joints [13.419, 59.512, 7.261, -144.32, 70.782, 166.702]
  Set speed (17.9 mm/s)
  Call Extruder(1218.37706)
  MoveL 4997 to (454.57, 546.76, 88) mm, rotated rx -180 ry 0 rz 160 deg; joints [13.334, 59.379, 7.564, -144.442, 70.9, 166.835]
  Set speed (17.9 mm/s)
  Call Extruder(1222.94949)
  MoveL 4998 to (453.54, 545.74, 88) mm, rotated rx -180 ry 0 rz 160 deg; joints [13.229, 59.224, 7.917, -144.59, 71.037, 166.992]
  Set speed (17.9 mm/s)
  Call Extruder(1227.15409)
  MoveL 4999 to (452.61, 544.77, 88) mm, rotated rx -180 ry 0 rz 160 deg; joints [13.128, 59.084, 8.236, -144.729, 71.161, 167.135]
  Set speed (18.0 mm/s)
  Call Extruder(1231.32233)
  MoveL 5000 to (451.71, 543.8, 88) mm, rotated rx -180 ry 0 rz 160 deg; joints [13.025, 58.948, 8.546, -144.87, 71.28, 167.275]
  Set speed (17.9 mm/s)
  Call Extruder(1234.68081)
  MoveL 5001 to (451, 543, 88) mm, rotated rx -180 ry 0 rz 160 deg; joints [12.939, 58.84, 8.792, -144.985, 71.375, 167.388]
  Set speed (17.9 mm/s)
  Call Extruder(1239.72619)
  MoveL 5002 to (449.95, 541.79, 88) mm, rotated rx 180 ry 0 rz 160 deg; joints [12.805, 58.681, 9.155, -145.162, 71.513, 167.555]
  Set speed (17.9 mm/s)
  Call Extruder(1243.90592)
  MoveL 5003 to (449.11, 540.76, 88) mm, rotated rx 180 ry 0 rz 160 deg; joints [12.691, 58.553, 9.449, -145.311, 71.625, 167.691]
  Call Extruder(1248.12144)
  MoveL 5004 to (448.28, 539.7, 88) mm, rotated rx -180 ry 0 rz 160 deg; joints [12.572, 58.427, 9.739, -145.464, 71.734, 167.828]
  Set speed (17.9 mm/s)
  Call Extruder(1252.30781)
  MoveL 5005 to (447.49, 538.64, 88) mm, rotated rx 180 ry 0 rz 160 deg; joints [12.449, 58.304, 10.021, -145.62, 71.84, 167.962]
  Set speed (17.9 mm/s)
  Call Extruder(1256.49667)
  MoveL 5006 to (446.71, 537.56, 88) mm, rotated rx 180 ry 0 rz 160 deg; joints [12.324, 58.185, 10.297, -145.778, 71.943, 168.095]
  Set speed (17.9 mm/s)
  Call Extruder(1260.67306)
  MoveL 5007 to (445.95, 536.46, 88) mm, rotated rx -180 ry 0 rz 160 deg; joints [12.196, 58.068, 10.566, -145.938, 72.043, 168.226]
  Set speed (17.9 mm/s)
  Call Extruder(1264.87765)
  MoveL 5008 to (445.21, 535.35, 88) mm, rotated rx 180 ry 0 rz 160 deg; joints [12.063, 57.953, 10.83, -146.101, 72.14, 168.356]
  Call Extruder(1269.14994)
  MoveL 5009 to (444.49, 534.2, 88) mm, rotated rx 180 ry 0 rz 160 deg; joints [11.924, 57.84, 11.092, -146.27, 72.236, 168.486]
  Call Extruder(1273.26380)
  MoveL 5010 to (443.82, 533.08, 88) mm, rotated rx 180 ry 0 rz 160 deg; joints [11.788, 57.734, 11.337, -146.436, 72.324, 168.61]
  Set speed (17.9 mm/s)
  Call Extruder(1277.53819)
  MoveL 5011 to (443.14, 531.9, 88) mm, rotated rx -180 ry 0 rz 160 deg; joints [11.642, 57.628, 11.584, -146.61, 72.413, 168.737]
  Set speed (17.9 mm/s)
  Call Extruder(1281.58149)
  MoveL 5012 to (442.52, 530.77, 88) mm, rotated rx 180 ry 0 rz 160 deg; joints [11.502, 57.53, 11.812, -146.777, 72.495, 168.855]
  Set speed (17.9 mm/s)
  Call Extruder(1285.84595)
  MoveL 5013 to (441.89, 529.57, 88) mm, rotated rx -180 ry 0 rz 160 deg; joints [11.351, 57.429, 12.046, -146.955, 72.577, 168.978]
  Call Extruder(1289.99024)
  MoveL 5014 to (441.31, 528.39, 88) mm, rotated rx 180 ry 0 rz 160 deg; joints [11.201, 57.335, 12.265, -147.131, 72.653, 169.095]
  Set speed (17.9 mm/s)
  Call Extruder(1294.31800)
  MoveL 5015 to (440.73, 527.14, 88) mm, rotated rx 180 ry 0 rz 160 deg; joints [11.041, 57.24, 12.486, -147.317, 72.729, 169.216]
  Set speed (17.9 mm/s)
  Call Extruder(1298.34067)
  MoveL 5016 to (440.2, 525.98, 88) mm, rotated rx -180 ry 0 rz 160 deg; joints [10.89, 57.154, 12.687, -147.491, 72.798, 169.326]
  Call Extruder(1302.72111)
  MoveL 5017 to (439.67, 524.69, 88) mm, rotated rx 180 ry 0 rz 160 deg; joints [10.723, 57.065, 12.895, -147.683, 72.868, 169.444]
  Call Extruder(1306.91633)
  MoveL 5018 to (439.17, 523.46, 88) mm, rotated rx -180 ry 0 rz 160 deg; joints [10.56, 56.982, 13.089, -147.868, 72.932, 169.555]
  Set speed (17.9 mm/s)
  Call Extruder(1311.11455)
  MoveL 5019 to (438.71, 522.21, 88) mm, rotated rx -180 ry 0 rz 160 deg; joints [10.394, 56.904, 13.273, -148.057, 72.991, 169.664]
  Set speed (17.9 mm/s)
  Call Extruder(1315.31148)
  MoveL 5020 to (438.26, 520.95, 88) mm, rotated rx -180 ry 0 rz 160 deg; joints [10.226, 56.827, 13.452, -148.246, 73.049, 169.771]
  Set speed (17.9 mm/s)
  Call Extruder(1323.71042)
  MoveL 5021 to (437.45, 518.41, 88) mm, rotated rx -180 ry 0 rz 160 deg; joints [9.881, 56.686, 13.785, -148.631, 73.151, 169.979]
  Set speed (17.9 mm/s)
  Call Extruder(1327.89564)
  MoveL 5022 to (437.1, 517.13, 88) mm, rotated rx 180 ry 0 rz 160 deg; joints [9.705, 56.621, 13.938, -148.826, 73.196, 170.079]
  Call Extruder(1332.05325)
  MoveL 5023 to (436.76, 515.85, 88) mm, rotated rx -180 ry 0 rz 160 deg; joints [9.53, 56.558, 14.085, -149.019, 73.238, 170.176]
  Set speed (17.9 mm/s)
  Call Extruder(1336.30166)
  MoveL 5024 to (436.45, 514.54, 88) mm, rotated rx -180 ry 0 rz 160 deg; joints [9.348, 56.499, 14.224, -149.219, 73.276, 170.273]
  Set speed (17.9 mm/s)
  Call Extruder(1340.44543)
  MoveL 5025 to (436.17, 513.25, 88) mm, rotated rx 180 ry 0 rz 160 deg; joints [9.168, 56.444, 14.355, -149.415, 73.311, 170.367]
  Set speed (17.9 mm/s)
  Call Extruder(1348.91489)
  MoveL 5026 to (435.67, 510.61, 88) mm, rotated rx 180 ry 0 rz 160 deg; joints [8.796, 56.342, 14.596, -149.82, 73.369, 170.55]
  Set speed (17.9 mm/s)
  Call Extruder(1357.30793)
  MoveL 5027 to (435.29, 507.97, 88) mm, rotated rx -180 ry 0 rz 160 deg; joints [8.42, 56.255, 14.801, -150.225, 73.41, 170.722]
  Set speed (17.9 mm/s)
  Call Extruder(1365.68630)
  MoveL 5028 to (435.02, 505.32, 88) mm, rotated rx -180 ry 0 rz 160 deg; joints [8.038, 56.182, 14.973, -150.632, 73.436, 170.886]
  Call Extruder(1373.93227)
  MoveL 5029 to (434.86, 502.7, 88) mm, rotated rx -180 ry 0 rz 160 deg; joints [7.659, 56.125, 15.11, -151.035, 73.445, 171.037]
  Set speed (17.9 mm/s)
  Call Extruder(1382.37731)
  MoveL 5030 to (434.8, 500.02, 88) mm, rotated rx -180 ry 0 rz 160 deg; joints [7.266, 56.079, 15.217, -151.448, 73.439, 171.184]
  Set speed (17.9 mm/s)
  Call Extruder(1390.01188)
  MoveL 5031 to (434.85, 497.59, 88) mm, rotated rx -180 ry 0 rz 160 deg; joints [6.909, 56.051, 15.285, -151.822, 73.419, 171.308]
  Call Extruder(1397.47719)
  MoveL 5032 to (434.98, 495.22, 88) mm, rotated rx 180 ry 0 rz 160 deg; joints [6.558, 56.034, 15.325, -152.188, 73.387, 171.423]
  Set speed (17.9 mm/s)
  Call Extruder(1405.01237)
  MoveL 5033 to (435.2, 492.83, 88) mm, rotated rx -180 ry 0 rz 160 deg; joints [6.203, 56.029, 15.336, -152.555, 73.34, 171.531]
  Set speed (17.9 mm/s)
  Call Extruder(1412.56965)
  MoveL 5034 to (435.51, 490.45, 88) mm, rotated rx -180 ry 0 rz 160 deg; joints [5.847, 56.035, 15.322, -152.921, 73.28, 171.633]
  Set speed (17.9 mm/s)
  Call Extruder(1420.19521)
  MoveL 5035 to (435.91, 488.05, 88) mm, rotated rx -180 ry 0 rz 160 deg; joints [5.488, 56.053, 15.279, -153.288, 73.206, 171.728]
  Set speed (17.9 mm/s)
  Call Extruder(1427.59516)
  MoveL 5036 to (436.38, 485.75, 88) mm, rotated rx -180 ry 0 rz 160 deg; joints [5.142, 56.082, 15.211, -153.641, 73.122, 171.813]
  Set speed (17.9 mm/s)
  Call Extruder(1435.21039)
  MoveL 5037 to (436.95, 483.4, 88) mm, rotated rx 180 ry 0 rz 160 deg; joints [4.788, 56.123, 15.114, -154, 73.021, 171.894]
  Call Extruder(1442.66983)
  MoveL 5038 to (437.6, 481.11, 88) mm, rotated rx -180 ry 0 rz 160 deg; joints [4.444, 56.175, 14.991, -154.346, 72.909, 171.966]
  Set speed (17.9 mm/s)
  Call Extruder(1450.22891)
  MoveL 5039 to (438.34, 478.83, 88) mm, rotated rx -180 ry 0 rz 160 deg; joints [4.1, 56.239, 14.84, -154.692, 72.782, 172.032]
  Call Extruder(1457.93850)
  MoveL 5040 to (439.18, 476.52, 88) mm, rotated rx 180 ry 0 rz 160 deg; joints [3.753, 56.315, 14.66, -155.038, 72.64, 172.093]
  Set speed (17.9 mm/s)
  Call Extruder(1465.47856)
  MoveL 5041 to (440.08, 474.3, 88) mm, rotated rx 180 ry 0 rz 160 deg; joints [3.418, 56.401, 14.456, -155.37, 72.487, 172.145]
  Set speed (17.9 mm/s)
  Call Extruder(1472.86605)
  MoveL 5042 to (441.05, 472.16, 88) mm, rotated rx -180 ry 0 rz 160 deg; joints [3.097, 56.496, 14.231, -155.687, 72.325, 172.19]
  Set speed (17.9 mm/s)
  Call Extruder(1480.53431)
  MoveL 5043 to (442.13, 469.97, 88) mm, rotated rx 180 ry 0 rz 160 deg; joints [2.769, 56.607, 13.971, -156.008, 72.144, 172.229]
  Call Extruder(1487.91809)
  MoveL 5044 to (443.25, 467.91, 88) mm, rotated rx 180 ry 0 rz 160 deg; joints [2.46, 56.723, 13.696, -156.309, 71.958, 172.261]
  Set speed (18.0 mm/s)
  Call Extruder(1495.66295)
  MoveL 5045 to (444.5, 465.79, 88) mm, rotated rx 180 ry 0 rz 160 deg; joints [2.144, 56.857, 13.382, -156.615, 71.75, 172.288]
  Set speed (18.0 mm/s)
  Call Extruder(1503.03002)
  MoveL 5046 to (445.77, 463.81, 88) mm, rotated rx -180 ry 0 rz 160 deg; joints [1.852, 56.995, 13.058, -156.897, 71.541, 172.307]
  Set speed (17.9 mm/s)
  Call Extruder(1510.67228)
  MoveL 5047 to (447.15, 461.82, 88) mm, rotated rx -180 ry 0 rz 160 deg; joints [1.557, 57.149, 12.699, -157.178, 71.312, 172.321]
  Call Extruder(1518.07484)
  MoveL 5048 to (448.57, 459.94, 88) mm, rotated rx 180 ry 0 rz 160 deg; joints [1.28, 57.308, 12.327, -157.439, 71.079, 172.327]
  Call Extruder(1525.61462)
  MoveL 5049 to (450.08, 458.07, 88) mm, rotated rx 180 ry 0 rz 160 deg; joints [1.008, 57.481, 11.925, -157.694, 70.831, 172.328]
  Set speed (17.9 mm/s)
  Call Extruder(1533.22289)
  MoveL 5050 to (451.67, 456.25, 88) mm, rotated rx 180 ry 0 rz 160 deg; joints [0.744, 57.665, 11.498, -157.94, 70.57, 172.322]
  Set speed (17.9 mm/s)
  Call Extruder(1540.95198)
  MoveL 5051 to (453.35, 454.46, 88) mm, rotated rx 180 ry 0 rz 160 deg; joints [0.486, 57.863, 11.04, -158.177, 70.294, 172.31]
  Set speed (17.9 mm/s)
  Call Extruder(1548.39637)
  MoveL 5052 to (455.03, 452.79, 88) mm, rotated rx -180 ry 0 rz 160 deg; joints [0.248, 58.063, 10.578, -158.392, 70.019, 172.292]
  Set speed (17.9 mm/s)
  Call Extruder(1555.99532)
  MoveL 5053 to (456.81, 451.16, 88) mm, rotated rx 180 ry 0 rz 160 deg; joints [0.016, 58.277, 10.084, -158.599, 69.727, 172.267]
  Set speed (17.9 mm/s)
  Call Extruder(1563.54265)
  MoveL 5054 to (458.64, 449.6, 88) mm, rotated rx 180 ry 0 rz 160 deg; joints [-0.202, 58.499, 9.573, -158.791, 69.429, 172.236]
  Set speed (17.9 mm/s)
  Call Extruder(1571.39618)
  MoveL 5055 to (460.6, 448.06, 88) mm, rotated rx -180 ry 0 rz 160 deg; joints [-0.418, 58.74, 9.022, -158.977, 69.11, 172.197]
  Call Extruder(0.00000)
  Set speed (17.9 mm/s)
  Call Extruder(6.66527)
  MoveL 5056 to (462.31, 446.8, 88) mm, rotated rx 180 ry 0 rz 160 deg; joints [-0.59, 58.952, 8.538, -159.123, 68.832, 172.158]
  Set speed (17.9 mm/s)
  Call Extruder(14.76548)
  MoveL 5057 to (464.44, 445.36, 88) mm, rotated rx 180 ry 0 rz 160 deg; joints [-0.787, 59.219, 7.929, -159.285, 68.486, 172.104]
  Set speed (17.9 mm/s)
  Call Extruder(22.39742)
  MoveL 5058 to (466.49, 444.07, 88) mm, rotated rx 180 ry 0 rz 160 deg; joints [-0.961, 59.479, 7.336, -159.423, 68.151, 172.046]
  Set speed (17.9 mm/s)
  Call Extruder(29.93934)
  MoveL 5059 to (468.57, 442.88, 88) mm, rotated rx -180 ry 0 rz 160 deg; joints [-1.12, 59.745, 6.733, -159.545, 67.814, 171.983]
  Set speed (17.9 mm/s)
  Call Extruder(38.34375)
  MoveL 5060 to (470.94, 441.64, 88) mm, rotated rx -180 ry 0 rz 160 deg; joints [-1.282, 60.051, 6.043, -159.664, 67.431, 171.904]
  Set speed (17.9 mm/s)
  Call Extruder(39.16815)
  MoveL 5061 to (471.18, 441.53, 88) mm, rotated rx 180 ry 0 rz 160 deg; joints [-1.296, 60.082, 5.973, -159.673, 67.392, 171.895]
  Set speed (17.9 mm/s)
  Call Extruder(45.04685)
  MoveL 5062 to (472.86, 440.72, 88) mm, rotated rx 180 ry 0 rz 160 deg; joints [-1.401, 60.302, 5.478, -159.745, 67.119, 171.835]
  Call Extruder(52.60034)
  MoveL 5063 to (475.06, 439.76, 88) mm, rotated rx 180 ry 0 rz 160 deg; joints [-1.523, 60.592, 4.827, -159.824, 66.763, 171.751]
  Set speed (17.9 mm/s)
  Call Extruder(60.06790)
  MoveL 5064 to (477.27, 438.89, 88) mm, rotated rx 180 ry 0 rz 160 deg; joints [-1.632, 60.886, 4.169, -159.887, 66.405, 171.661]
  Set speed (17.9 mm/s)
  Call Extruder(67.70269)
  MoveL 5065 to (479.56, 438.09, 88) mm, rotated rx 180 ry 0 rz 160 deg; joints [-1.73, 61.193, 3.482, -159.936, 66.035, 171.562]
  Set speed (17.9 mm/s)
  Call Extruder(75.09503)
  MoveL 5066 to (481.81, 437.39, 88) mm, rotated rx -180 ry 0 rz 160 deg; joints [-1.814, 61.497, 2.805, -159.969, 65.672, 171.458]
  Call Extruder(82.58260)
  MoveL 5067 to (484.11, 436.77, 88) mm, rotated rx -180 ry 0 rz 160 deg; joints [-1.886, 61.812, 2.107, -159.988, 65.301, 171.347]
  Set speed (17.9 mm/s)
  Call Extruder(90.34294)
  MoveL 5068 to (486.51, 436.21, 88) mm, rotated rx 180 ry 0 rz 160 deg; joints [-1.949, 62.144, 1.372, -159.993, 64.913, 171.224]
  Set speed (17.9 mm/s)
  Call Extruder(97.74689)
  MoveL 5069 to (488.82, 435.77, 88) mm, rotated rx 180 ry 0 rz 160 deg; joints [-1.997, 62.467, 0.66, -159.982, 64.54, 171.099]
  Set speed (18.0 mm/s)
  Call Extruder(105.39773)
  MoveL 5070 to (491.23, 435.39, 88) mm, rotated rx -180 ry 0 rz 160 deg; joints [-2.034, 62.805, -0.086, -159.956, 64.151, 170.962]
  Call Extruder(112.93155)
  MoveL 5071 to (493.61, 435.12, 88) mm, rotated rx 180 ry 0 rz 160 deg; joints [-2.059, 63.144, -0.829, -159.916, 63.768, 170.819]
  Set speed (17.9 mm/s)
  Call Extruder(120.36281)
  MoveL 5072 to (495.97, 434.93, 88) mm, rotated rx 180 ry 0 rz 160 deg; joints [-2.073, 63.483, -1.57, -159.862, 63.388, 170.672]
  Set speed (17.9 mm/s)
  Call Extruder(128.06762)
  MoveL 5073 to (498.41, 434.82, 88) mm, rotated rx 180 ry 0 rz 160 deg; joints [-2.075, 63.839, -2.346, -159.791, 62.993, 170.51]
  Call Extruder(135.54540)
  MoveL 5074 to (500.79, 434.81, 88) mm, rotated rx -180 ry 0 rz 160 deg; joints [-2.066, 64.188, -3.105, -159.708, 62.609, 170.346]
  Set speed (17.9 mm/s)
  Call Extruder(143.16046)
  MoveL 5075 to (503.21, 434.88, 88) mm, rotated rx 180 ry 0 rz 160 deg; joints [-2.045, 64.547, -3.885, -159.609, 62.219, 170.171]
  Set speed (18.0 mm/s)
  Call Extruder(150.63276)
  MoveL 5076 to (505.59, 435.04, 88) mm, rotated rx -180 ry 0 rz 160 deg; joints [-2.015, 64.903, -4.654, -159.498, 61.836, 169.991]
  Set speed (17.9 mm/s)
  Call Extruder(158.26149)
  MoveL 5077 to (508, 435.3, 88) mm, rotated rx 180 ry 0 rz 160 deg; joints [-1.972, 65.269, -5.444, -159.37, 61.447, 169.799]
  Set speed (17.9 mm/s)
  Call Extruder(165.65593)
  MoveL 5078 to (510.33, 435.63, 88) mm, rotated rx -180 ry 0 rz 160 deg; joints [-1.921, 65.626, -6.212, -159.233, 61.072, 169.606]
  Set speed (17.9 mm/s)
  Call Extruder(173.27014)
  MoveL 5079 to (512.71, 436.05, 88) mm, rotated rx 180 ry 0 rz 160 deg; joints [-1.858, 65.995, -7.006, -159.078, 60.687, 169.399]
  Set speed (17.9 mm/s)
  Call Extruder(180.14758)
  MoveL 5080 to (514.84, 436.52, 88) mm, rotated rx 180 ry 0 rz 160 deg; joints [-1.793, 66.33, -7.723, -158.927, 60.342, 169.205]
  Set speed (17.9 mm/s)
  Call Extruder(188.30625)
  MoveL 5081 to (517.36, 437.16, 88) mm, rotated rx 180 ry 0 rz 160 deg; joints [-1.705, 66.729, -8.575, -158.733, 59.936, 168.967]
  Set speed (17.9 mm/s)
  Call Extruder(195.93449)
  MoveL 5082 to (519.68, 437.84, 88) mm, rotated rx -180 ry 0 rz 160 deg; joints [-1.612, 67.103, -9.371, -158.538, 59.56, 168.735]
  Set speed (18.0 mm/s)
  Call Extruder(203.55142)
  MoveL 5083 to (521.98, 438.62, 88) mm, rotated rx 180 ry 0 rz 160 deg; joints [-1.51, 67.476, -10.166, -158.331, 59.189, 168.497]
  Set speed (18.0 mm/s)
  Call Extruder(211.01298)
  MoveL 5084 to (524.2, 439.46, 88) mm, rotated rx 180 ry 0 rz 160 deg; joints [-1.401, 67.842, -10.941, -158.115, 58.83, 168.255]
  Set speed (17.9 mm/s)
  Call Extruder(218.63554)
  MoveL 5085 to (526.43, 440.4, 88) mm, rotated rx 180 ry 0 rz 160 deg; joints [-1.281, 68.215, -11.73, -157.882, 58.469, 168.001]
  Call Extruder(226.09742)
  MoveL 5086 to (528.58, 441.4, 88) mm, rotated rx -180 ry 0 rz 160 deg; joints [-1.156, 68.579, -12.499, -157.644, 58.121, 167.745]
  Call Extruder(233.73094)
  MoveL 5087 to (530.75, 442.51, 88) mm, rotated rx 180 ry 0 rz 160 deg; joints [-1.019, 68.949, -13.279, -157.387, 57.772, 167.476]
  Call Extruder(241.28187)
  MoveL 5088 to (532.84, 443.68, 88) mm, rotated rx -180 ry 0 rz 160 deg; joints [-0.875, 69.313, -14.045, -157.123, 57.433, 167.204]
  Set speed (17.9 mm/s)
  Call Extruder(248.74625)
  MoveL 5089 to (534.87, 444.91, 88) mm, rotated rx 180 ry 0 rz 160 deg; joints [-0.726, 69.671, -14.795, -156.851, 57.105, 166.928]
  Set speed (17.9 mm/s)
  Call Extruder(256.37657)
  MoveL 5090 to (536.9, 446.25, 88) mm, rotated rx 180 ry 0 rz 160 deg; joints [-0.565, 70.033, -15.552, -156.563, 56.778, 166.639]
  Call Extruder(263.83359)
  MoveL 5091 to (538.83, 447.63, 88) mm, rotated rx -180 ry 0 rz 160 deg; joints [-0.401, 70.383, -16.284, -156.271, 56.467, 166.351]
  Call Extruder(271.29355)
  MoveL 5092 to (540.71, 449.07, 88) mm, rotated rx -180 ry 0 rz 160 deg; joints [-0.23, 70.728, -17.005, -155.971, 56.165, 166.058]
  Set speed (17.9 mm/s)
  Call Extruder(279.06350)
  MoveL 5093 to (542.61, 450.65, 88) mm, rotated rx -180 ry 0 rz 160 deg; joints [-0.046, 71.083, -17.744, -155.648, 55.859, 165.748]
  Set speed (17.9 mm/s)
  Call Extruder(286.52244)
  MoveL 5094 to (544.38, 452.23, 88) mm, rotated rx -180 ry 0 rz 160 deg; joints [0.138, 71.419, -18.442, -155.331, 55.576, 165.445]
  Set speed (18.0 mm/s)
  Call Extruder(294.08954)
  MoveL 5095 to (546.11, 453.9, 88) mm, rotated rx -180 ry 0 rz 160 deg; joints [0.331, 71.753, -19.135, -155.001, 55.298, 165.133]
  Set speed (17.9 mm/s)
  Call Extruder(298.18112)
  MoveL 5096 to (547.02, 454.83, 88) mm, rotated rx 180 ry 0 rz 160 deg; joints [0.438, 71.931, -19.503, -154.819, 55.154, 164.963]
  Set speed (17.9 mm/s)
  Call Extruder(302.33107)
  MoveL 5097 to (547.92, 455.8, 88) mm, rotated rx 180 ry 0 rz 160 deg; joints [0.548, 72.109, -19.872, -154.632, 55.01, 164.79]
  Set speed (17.9 mm/s)
  Call Extruder(306.61019)
  MoveL 5098 to (548.83, 456.81, 88) mm, rotated rx -180 ry 0 rz 160 deg; joints [0.663, 72.291, -20.248, -154.438, 54.865, 164.61]
  Set speed (17.9 mm/s)
  Call Extruder(310.75209)
  MoveL 5099 to (549.7, 457.8, 88) mm, rotated rx 180 ry 0 rz 160 deg; joints [0.776, 72.463, -20.605, -154.248, 54.729, 164.435]
  Set speed (17.9 mm/s)
  Call Extruder(314.91432)
  MoveL 5100 to (550.54, 458.82, 88) mm, rotated rx 180 ry 0 rz 160 deg; joints [0.891, 72.635, -20.96, -154.056, 54.596, 164.259]
  Set speed (17.9 mm/s)
  Call Extruder(319.92491)
  MoveL 5101 to (551.54, 460.07, 88) mm, rotated rx -180 ry 0 rz 160 deg; joints [1.032, 72.839, -21.379, -153.822, 54.44, 164.045]
  Set speed (17.9 mm/s)
  Call Extruder(323.32293)
  MoveL 5102 to (552.19, 460.92, 88) mm, rotated rx 180 ry 0 rz 160 deg; joints [1.129, 72.975, -21.659, -153.662, 54.337, 163.9]
  Call Extruder(327.51724)
  MoveL 5103 to (552.98, 462, 88) mm, rotated rx 180 ry 0 rz 160 deg; joints [1.25, 73.139, -21.998, -153.463, 54.215, 163.721]
  Call Extruder(331.73523)
  MoveL 5104 to (553.75, 463.1, 88) mm, rotated rx -180 ry 0 rz 160 deg; joints [1.373, 73.302, -22.333, -153.261, 54.096, 163.54]
  Set speed (17.9 mm/s)
  Call Extruder(335.97206)
  MoveL 5105 to (554.5, 464.22, 88) mm, rotated rx 180 ry 0 rz 160 deg; joints [1.498, 73.462, -22.663, -153.057, 53.98, 163.359]
  Set speed (17.9 mm/s)
  Call Extruder(340.10035)
  MoveL 5106 to (555.21, 465.32, 88) mm, rotated rx 180 ry 0 rz 160 deg; joints [1.621, 73.616, -22.978, -152.858, 53.871, 163.182]
  Set speed (17.9 mm/s)
  Call Extruder(344.35761)
  MoveL 5107 to (555.92, 466.48, 88) mm, rotated rx -180 ry 0 rz 160 deg; joints [1.75, 73.77, -23.296, -152.651, 53.764, 162.999]
  Set speed (17.9 mm/s)
  Call Extruder(348.53272)
  MoveL 5108 to (556.59, 467.62, 88) mm, rotated rx 180 ry 0 rz 160 deg; joints [1.877, 73.919, -23.6, -152.447, 53.663, 162.821]
  Set speed (17.9 mm/s)
  Call Extruder(353.95859)
  MoveL 5109 to (557.43, 469.13, 88) mm, rotated rx -180 ry 0 rz 160 deg; joints [2.044, 74.106, -23.985, -152.181, 53.538, 162.589]
  Set speed (17.9 mm/s)
  Call Extruder(356.91184)
  MoveL 5110 to (557.86, 469.96, 88) mm, rotated rx -180 ry 0 rz 160 deg; joints [2.136, 74.205, -24.188, -152.036, 53.473, 162.464]
  Set speed (17.9 mm/s)
  Call Extruder(361.06542)
  MoveL 5111 to (558.46, 471.14, 88) mm, rotated rx -180 ry 0 rz 160 deg; joints [2.266, 74.343, -24.469, -151.832, 53.386, 162.288]
  Set speed (17.9 mm/s)
  Call Extruder(365.28773)
  MoveL 5112 to (559.04, 472.35, 88) mm, rotated rx -180 ry 0 rz 160 deg; joints [2.4, 74.478, -24.747, -151.623, 53.302, 162.109]
  Set speed (17.9 mm/s)
  Call Extruder(369.54579)
